C03640=1069.715,413.514,387.232,175.844,35.074,156.512
C03641=1069.725,413.793,387.183,175.850,35.085,156.515
C03642=1069.734,414.072,387.133,175.857,35.096,156.518
C03643=1069.742,414.350,387.084,175.864,35.108,156.520
C03644=1069.751,414.596,387.041,175.870,35.117,156.523
C03645=1069.759,414.842,386.997,175.877,35.127,156.525
C03646=1069.766,415.088,386.953,175.883,35.137,156.527
C03647=1069.774,415.334,386.909,175.888,35.147,156.530
C03648=1069.782,415.580,386.865,175.894,35.157,156.532
C03649=1069.789,415.826,386.822,175.901,35.167,156.535
C03650=1069.797,416.072,386.778,175.907,35.177,156.537
C03651=1069.804,416.319,386.733,175.913,35.187,156.539
C03652=1069.813,416.564,386.689,175.919,35.197,156.542
C03653=1069.820,416.811,386.646,175.926,35.208,156.544
C03654=1069.828,417.056,386.601,175.932,35.218,156.547
C03655=1069.836,417.302,386.557,175.938,35.228,156.549
C03656=1069.844,417.549,386.513,175.944,35.238,156.552
C03657=1069.852,417.794,386.469,175.951,35.248,156.554
C03658=1069.860,418.040,386.425,175.957,35.259,156.557
C03659=1069.868,418.286,386.380,175.963,35.269,156.559
C03660=1069.875,418.532,386.336,175.970,35.279,156.562
C03661=1069.883,418.778,386.292,175.976,35.290,156.564
C03662=1069.892,419.024,386.247,175.983,35.300,156.567
C03663=1069.900,419.270,386.203,175.989,35.310,156.569
C03664=1069.908,419.515,386.159,175.995,35.321,156.572
C03665=1069.916,419.761,386.114,176.003,35.331,156.574
C03666=1069.924,420.007,386.070,176.009,35.342,156.577
C03667=1069.932,420.254,386.025,176.016,35.353,156.579
C03668=1069.940,420.499,385.980,176.022,35.363,156.582
C03669=1069.948,420.745,385.936,176.029,35.373,156.584
C03670=1069.956,420.991,385.892,176.035,35.384,156.587
C03671=1069.964,421.238,385.846,176.042,35.395,156.590
C03672=1069.972,421.483,385.801,176.048,35.406,156.592
C03673=1069.980,421.729,385.757,176.055,35.417,156.595
C03674=1069.988,421.975,385.712,176.062,35.427,156.598
C03675=1069.996,422.220,385.667,176.069,35.438,156.600
C03676=1070.004,422.466,385.622,176.075,35.449,156.603
C03677=1070.012,422.712,385.577,176.082,35.460,156.606
C03678=1070.020,422.957,385.532,176.088,35.471,156.608
C03679=1070.028,423.203,385.487,176.095,35.482,156.611
C03680=1070.037,423.449,385.442,176.102,35.493,156.614
C03681=1070.044,423.695,385.396,176.109,35.504,156.616
C03682=1070.052,423.940,385.352,176.115,35.515,156.619
C03683=1070.061,424.187,385.306,176.122,35.526,156.622
C03684=1070.069,424.432,385.261,176.130,35.537,156.625
C03685=1070.076,424.678,385.216,176.136,35.548,156.627
C03686=1070.085,424.924,385.171,176.143,35.559,156.630
C03687=1070.093,425.169,385.125,176.150,35.571,156.633
C03688=1070.102,425.415,385.080,176.157,35.582,156.636
C03689=1070.110,425.660,385.034,176.164,35.593,156.638
C03690=1070.118,425.907,384.989,176.171,35.604,156.641
C03691=1070.126,426.152,384.944,176.177,35.615,156.644
C03692=1070.135,426.398,384.898,176.185,35.627,156.647
C03693=1070.143,426.643,384.852,176.192,35.638,156.650
C03694=1070.152,426.889,384.807,176.199,35.650,156.652
C03695=1070.159,427.135,384.761,176.206,35.661,156.655
C03696=1070.170,427.431,384.706,176.214,35.675,156.659
C03697=1070.179,427.729,384.650,176.223,35.689,156.662
C03698=1070.190,428.026,384.595,176.232,35.703,156.666
C03699=1070.199,428.324,384.539,176.240,35.717,156.669
C03700=1070.208,428.570,384.493,176.248,35.729,156.672
C03701=1070.217,428.815,384.447,176.255,35.741,156.675
C03702=1070.224,429.061,384.401,176.263,35.753,156.678
C03703=1070.233,429.306,384.355,176.270,35.764,156.681
C03704=1070.241,429.552,384.309,176.277,35.776,156.684
C03705=1070.250,429.797,384.263,176.285,35.788,156.687
C03706=1070.258,430.043,384.217,176.291,35.800,156.690
C03707=1070.267,430.288,384.170,176.299,35.812,156.693
C03708=1070.275,430.534,384.123,176.306,35.824,156.696
C03709=1070.283,430.779,384.078,176.314,35.836,156.699
C03710=1070.292,431.025,384.032,176.321,35.848,156.702
C03711=1070.301,431.270,383.985,176.329,35.860,156.705
C03712=1070.309,431.516,383.939,176.336,35.872,156.708
C03713=1070.318,431.762,383.892,176.344,35.884,156.711
C03714=1070.326,432.007,383.845,176.352,35.896,156.714
C03715=1070.334,432.252,383.799,176.359,35.909,156.717
C03716=1070.343,432.498,383.752,176.367,35.922,156.721
C03717=1070.351,432.743,383.706,176.374,35.934,156.724
C03718=1070.360,432.989,383.659,176.382,35.946,156.727
C03719=1070.368,433.234,383.612,176.390,35.959,156.730
C03720=1070.377,433.479,383.565,176.397,35.971,156.733
C03721=1070.386,433.725,383.518,176.406,35.984,156.736
C03722=1070.393,433.970,383.471,176.414,35.996,156.739
C03723=1070.402,434.216,383.424,176.421,36.009,156.743
C03724=1070.411,434.461,383.377,176.429,36.021,156.746
C03725=1070.419,434.706,383.330,176.437,36.034,156.749
C03726=1070.428,434.952,383.283,176.444,36.047,156.752
C03727=1070.437,435.197,383.236,176.452,36.059,156.756
C03728=1070.445,435.442,383.189,176.461,36.072,156.759
C03729=1070.454,435.687,383.141,176.468,36.085,156.762
C03730=1070.463,435.933,383.095,176.476,36.098,156.765
C03731=1070.471,436.178,383.047,176.484,36.111,156.769
C03732=1070.480,436.423,382.999,176.493,36.124,156.772
C03733=1070.489,436.669,382.952,176.501,36.137,156.775
C03734=1070.498,436.914,382.905,176.508,36.150,156.779
C03735=1070.506,437.159,382.857,176.516,36.163,156.782
C03736=1070.515,437.404,382.810,176.525,36.176,156.785
C03737=1070.525,437.649,382.762,176.533,36.189,156.789
C03738=1070.533,437.894,382.714,176.541,36.202,156.792
C03739=1070.541,438.140,382.667,176.550,36.215,156.796
C03740=1070.551,438.386,382.619,176.558,36.229,156.799
C03741=1070.560,438.630,382.572,176.566,36.242,156.802
C03742=1070.568,438.875,382.523,176.574,36.255,156.806
C03743=1070.578,439.121,382.475,176.582,36.269,156.809
C03744=1070.586,439.365,382.428,176.591,36.282,156.813
C03745=1070.595,439.611,382.380,176.599,36.295,156.816
C03746=1070.604,439.856,382.332,176.608,36.309,156.820
C03747=1070.612,440.101,382.283,176.616,36.323,156.823
C03748=1070.622,440.346,382.236,176.625,36.336,156.827
C03749=1070.631,440.591,382.188,176.633,36.350,156.830
C03750=1070.640,440.837,382.139,176.642,36.364,156.834
C03751=1070.649,441.082,382.092,176.650,36.377,156.838
C03752=1070.657,441.314,382.045,176.659,36.391,156.841
C03753=1070.665,441.548,381.999,176.667,36.404,156.845
C03754=1070.674,441.781,381.953,176.675,36.417,156.848
C03755=1070.683,442.015,381.907,176.683,36.430,156.851
C03756=1070.692,442.248,381.860,176.693,36.444,156.855
C03757=1070.700,442.481,381.814,176.701,36.457,156.858
C03758=1070.708,442.715,381.768,176.709,36.471,156.862
C03759=1070.717,442.948,381.721,176.718,36.484,156.865
C03760=1070.727,443.193,381.673,176.726,36.498,156.869
C03761=1070.736,443.438,381.624,176.735,36.513,156.873
C03762=1070.745,443.682,381.575,176.744,36.527,156.877
C03763=1070.754,443.927,381.526,176.754,36.541,156.881
C03764=1070.764,444.172,381.478,176.762,36.556,156.884
C03765=1070.773,444.418,381.429,176.771,36.570,156.888
C03766=1070.781,444.662,381.380,176.781,36.584,156.892
C03767=1070.790,444.908,381.331,176.790,36.599,156.896
C03768=1070.800,445.152,381.281,176.799,36.614,156.900
C03769=1070.809,445.397,381.232,176.808,36.628,156.904
C03770=1070.819,445.642,381.183,176.817,36.643,156.907
C03771=1070.828,445.887,381.133,176.826,36.658,156.911
C03772=1070.837,446.132,381.085,176.836,36.672,156.915
C03773=1070.846,446.376,381.035,176.845,36.687,156.919
C03774=1070.855,446.621,380.986,176.855,36.702,156.923
C03775=1070.864,446.866,380.936,176.864,36.717,156.927
C03776=1070.874,447.111,380.887,176.874,36.732,156.931
C03777=1070.884,447.355,380.837,176.883,36.747,156.935
C03778=1070.893,447.601,380.788,176.893,36.762,156.939
C03779=1070.903,447.846,380.738,176.902,36.777,156.943
C03780=1070.913,448.089,380.688,176.911,36.793,156.947
C03781=1070.922,448.332,380.640,176.920,36.807,156.951
C03782=1070.932,448.577,380.590,176.929,36.822,156.955
C03783=1070.944,448.821,380.542,176.937,36.836,156.959
C03784=1070.957,449.066,380.495,176.945,36.850,156.963
C03785=1070.972,449.311,380.449,176.953,36.863,156.966
C03786=1070.987,449.556,380.402,176.960,36.876,156.970
C03787=1071.004,449.802,380.357,176.968,36.888,156.973
C03788=1070.654,449.802,380.106,176.954,37.029,157.010
C03789=1070.638,449.556,380.151,176.947,37.016,157.007
C03790=1070.622,449.311,380.197,176.939,37.004,157.004
C03791=1070.608,449.066,380.244,176.931,36.990,157.000
C03792=1070.595,448.821,380.291,176.923,36.977,156.996
C03793=1070.582,448.576,380.339,176.914,36.963,156.993
C03794=1070.571,448.332,380.388,176.905,36.948,156.989
C03795=1070.562,448.088,380.437,176.896,36.933,156.985
C03796=1070.553,447.845,380.487,176.886,36.918,156.981
C03797=1070.543,447.601,380.537,176.877,36.903,156.977
C03798=1070.533,447.356,380.587,176.867,36.888,156.973
C03799=1070.523,447.111,380.636,176.858,36.873,156.969
C03800=1070.514,446.866,380.685,176.848,36.858,156.965
C03801=1070.505,446.621,380.735,176.838,36.843,156.961
C03802=1070.496,446.376,380.785,176.829,36.828,156.957
C03803=1070.486,446.131,380.834,176.819,36.814,156.953
C03804=1070.477,445.887,380.884,176.810,36.799,156.949
C03805=1070.468,445.641,380.933,176.800,36.784,156.945
C03806=1070.458,445.397,380.982,176.792,36.770,156.941
C03807=1070.449,445.153,381.031,176.782,36.755,156.937
C03808=1070.440,444.908,381.080,176.773,36.741,156.933
C03809=1070.431,444.663,381.130,176.764,36.726,156.929
C03810=1070.422,444.417,381.179,176.754,36.711,156.925
C03811=1070.412,444.173,381.228,176.745,36.697,156.922
C03812=1070.403,443.928,381.277,176.736,36.683,156.918
C03813=1070.394,443.683,381.326,176.727,36.668,156.914
C03814=1070.384,443.438,381.374,176.718,36.654,156.910
C03815=1070.375,443.193,381.423,176.708,36.640,156.906
C03816=1070.366,442.949,381.472,176.700,36.626,156.903
C03817=1070.358,442.724,381.516,176.692,36.612,156.899
C03818=1070.349,442.500,381.561,176.684,36.600,156.896
C03819=1070.341,442.276,381.606,176.675,36.587,156.892
C03820=1070.333,442.052,381.649,176.667,36.574,156.889
C03821=1070.324,441.828,381.694,176.659,36.562,156.886
C03822=1070.316,441.604,381.739,176.651,36.549,156.882
C03823=1070.308,441.380,381.782,176.643,36.536,156.879
C03824=1070.300,441.156,381.827,176.635,36.524,156.876
C03825=1070.291,440.912,381.876,176.627,36.510,156.872
C03826=1070.282,440.666,381.924,176.618,36.496,156.869
C03827=1070.273,440.421,381.973,176.609,36.482,156.865
C03828=1070.264,440.176,382.020,176.600,36.468,156.861
C03829=1070.254,439.931,382.069,176.592,36.455,156.858
C03830=1070.246,439.686,382.117,176.583,36.442,156.854
C03831=1070.237,439.441,382.164,176.575,36.428,156.851
C03832=1070.228,439.195,382.213,176.566,36.415,156.847
C03833=1070.219,438.951,382.261,176.558,36.401,156.844
C03834=1070.210,438.705,382.308,176.549,36.388,156.840
C03835=1070.202,438.460,382.357,176.541,36.374,156.837
C03836=1070.193,438.215,382.404,176.533,36.361,156.833
C03837=1070.183,437.969,382.452,176.524,36.348,156.830
C03838=1070.174,437.724,382.499,176.516,36.335,156.827
C03839=1070.166,437.480,382.547,176.507,36.322,156.823
C03840=1070.157,437.234,382.595,176.499,36.309,156.820
C03841=1070.148,436.989,382.643,176.491,36.296,156.817
C03842=1070.139,436.744,382.690,176.483,36.283,156.813
C03843=1070.130,436.498,382.737,176.475,36.270,156.810
C03844=1070.121,436.253,382.785,176.467,36.257,156.807
C03845=1070.112,436.008,382.832,176.459,36.244,156.803
C03846=1070.104,435.762,382.879,176.450,36.231,156.800
C03847=1070.096,435.517,382.927,176.442,36.218,156.797
C03848=1070.087,435.272,382.974,176.434,36.205,156.793
C03849=1070.078,435.027,383.021,176.427,36.193,156.790
C03850=1070.069,434.781,383.069,176.419,36.180,156.787
C03851=1070.060,434.536,383.115,176.410,36.167,156.784
C03852=1070.051,434.291,383.163,176.402,36.155,156.780
C03853=1070.043,434.045,383.210,176.395,36.142,156.777
C03854=1070.034,433.800,383.256,176.387,36.130,156.774
C03855=1070.026,433.554,383.303,176.379,36.117,156.771
C03856=1070.017,433.309,383.351,176.371,36.105,156.768
C03857=1070.008,433.064,383.397,176.364,36.092,156.764
C03858=1070.001,432.818,383.445,176.356,36.080,156.761
C03859=1069.992,432.572,383.491,176.348,36.068,156.758
C03860=1069.984,432.328,383.538,176.341,36.055,156.755
C03861=1069.976,432.082,383.584,176.333,36.043,156.752
C03862=1069.967,431.837,383.631,176.325,36.031,156.749
C03863=1069.958,431.591,383.678,176.318,36.018,156.746
C03864=1069.950,431.346,383.725,176.310,36.006,156.743
C03865=1069.941,431.100,383.771,176.303,35.994,156.740
C03866=1069.932,430.855,383.817,176.295,35.982,156.737
C03867=1069.924,430.609,383.863,176.287,35.970,156.734
C03868=1069.916,430.364,383.910,176.280,35.958,156.730
C03869=1069.907,430.118,383.957,176.272,35.946,156.727
C03870=1069.898,429.873,384.002,176.265,35.934,156.724
C03871=1069.890,429.627,384.049,176.257,35.923,156.721
C03872=1069.882,429.382,384.095,176.250,35.910,156.718
C03873=1069.874,429.136,384.141,176.242,35.899,156.716
C03874=1069.865,428.891,384.188,176.235,35.887,156.713
C03875=1069.857,428.645,384.233,176.228,35.875,156.710
C03876=1069.849,428.399,384.279,176.221,35.864,156.707
C03877=1069.838,428.100,384.335,176.212,35.849,156.703
C03878=1069.829,427.801,384.391,176.203,35.835,156.700
C03879=1069.818,427.503,384.447,176.194,35.821,156.696
C03880=1069.808,427.203,384.503,176.185,35.807,156.693
C03881=1069.800,426.957,384.549,176.178,35.796,156.690
C03882=1069.791,426.712,384.594,176.171,35.784,156.687
C03883=1069.783,426.466,384.640,176.164,35.773,156.684
C03884=1069.775,426.220,384.685,176.156,35.761,156.681
C03885=1069.766,425.974,384.731,176.150,35.750,156.678
C03886=1069.758,425.729,384.776,176.142,35.739,156.676
C03887=1069.750,425.483,384.822,176.135,35.728,156.673
C03888=1069.741,425.238,384.867,176.129,35.716,156.670
C03889=1069.733,424.992,384.913,176.121,35.705,156.667
C03890=1069.725,424.747,384.958,176.114,35.694,156.665
C03891=1069.717,424.501,385.004,176.108,35.683,156.662
C03892=1069.709,424.255,385.049,176.101,35.672,156.659
C03893=1069.701,424.009,385.094,176.093,35.661,156.656
C03894=1069.692,423.764,385.140,176.087,35.650,156.654
C03895=1069.685,423.517,385.185,176.080,35.639,156.651
C03896=1069.676,423.272,385.230,176.073,35.628,156.648
C03897=1069.667,423.027,385.275,176.066,35.617,156.645
C03898=1069.660,422.780,385.320,176.060,35.606,156.643
C03899=1069.652,422.535,385.365,176.053,35.595,156.640
C03900=1069.644,422.289,385.410,176.045,35.584,156.637
C03901=1069.635,422.043,385.455,176.039,35.573,156.635
C03902=1069.628,421.797,385.500,176.032,35.563,156.632
C03903=1069.620,421.552,385.545,176.026,35.552,156.629
C03904=1069.611,421.306,385.590,176.019,35.541,156.627
C03905=1069.604,421.060,385.635,176.012,35.530,156.624
C03906=1069.595,420.814,385.679,176.005,35.520,156.622
C03907=1069.587,420.568,385.724,175.999,35.509,156.619
C03908=1069.579,420.322,385.768,175.993,35.499,156.616
C03909=1069.571,420.076,385.813,175.986,35.488,156.614
C03910=1069.563,419.831,385.858,175.980,35.477,156.611
C03911=1069.555,419.585,385.903,175.973,35.467,156.609
C03912=1069.547,419.339,385.947,175.966,35.457,156.606
C03913=1069.539,419.093,385.991,175.959,35.446,156.604
C03914=1069.530,418.846,386.035,175.953,35.436,156.601
C03915=1069.522,418.601,386.080,175.947,35.426,156.599
C03916=1069.515,418.355,386.125,175.940,35.416,156.596
C03917=1069.507,418.109,386.169,175.934,35.405,156.594
C03918=1069.499,417.863,386.213,175.928,35.395,156.591
C03919=1069.491,417.617,386.258,175.921,35.384,156.589
C03920=1069.483,417.371,386.301,175.915,35.374,156.586
C03921=1069.475,417.125,386.346,175.909,35.364,156.584
C03922=1069.467,416.879,386.390,175.902,35.354,156.581
C03923=1069.459,416.633,386.434,175.896,35.344,156.579
C03924=1069.451,416.387,386.478,175.890,35.334,156.576
C03925=1069.444,416.141,386.523,175.883,35.323,156.574
C03926=1069.437,415.896,386.566,175.876,35.313,156.571
C03927=1069.429,415.650,386.610,175.870,35.304,156.569
C03928=1069.421,415.404,386.654,175.864,35.293,156.567
C03929=1069.413,415.158,386.698,175.859,35.284,156.564
C03930=1069.405,414.911,386.742,175.851,35.274,156.562
C03931=1069.397,414.665,386.786,175.846,35.264,156.560
C03932=1069.389,414.419,386.830,175.840,35.254,156.557
C03933=1069.380,414.139,386.879,175.832,35.243,156.554
C03934=1069.371,413.859,386.929,175.825,35.232,156.552
C03935=1069.362,413.579,386.979,175.818,35.220,156.549
C03936=1069.353,413.298,387.028,175.811,35.210,156.546
C03937=1069.346,413.053,387.072,175.805,35.200,156.544
C03938=1069.337,412.807,387.115,175.799,35.190,156.542
C03939=1069.329,412.561,387.158,175.793,35.180,156.540
C03940=1069.322,412.314,387.202,175.788,35.171,156.537
C03941=1069.314,412.069,387.245,175.782,35.162,156.535
C03942=1069.306,411.823,387.288,175.776,35.152,156.533
C03943=1069.298,411.576,387.332,175.770,35.142,156.530
C03944=1069.290,411.330,387.375,175.764,35.133,156.528
C03945=1069.284,411.084,387.418,175.757,35.123,156.526
C03946=1069.275,410.838,387.461,175.751,35.113,156.524
C03947=1069.267,410.591,387.505,175.745,35.104,156.521
C03948=1069.260,410.346,387.548,175.740,35.095,156.519
C03949=1069.252,410.099,387.591,175.734,35.085,156.517
C03950=1069.245,409.853,387.633,175.728,35.076,156.515
C03951=1069.237,409.607,387.677,175.722,35.067,156.513
C03952=1069.230,409.361,387.720,175.716,35.057,156.510
C03953=1069.222,409.115,387.763,175.710,35.048,156.508
C03954=1069.214,408.868,387.806,175.704,35.039,156.506
C03955=1069.207,408.622,387.849,175.699,35.030,156.504
C03956=1069.199,408.376,387.892,175.693,35.020,156.502
C03957=1069.191,408.130,387.935,175.687,35.011,156.499
C03958=1069.184,407.884,387.977,175.682,35.002,156.497
C03959=1069.176,407.637,388.020,175.676,34.993,156.495
C03960=1069.169,407.392,388.063,175.671,34.984,156.493
C03961=1069.161,407.145,388.105,175.665,34.975,156.491
C03962=1069.154,406.899,388.149,175.659,34.966,156.489
C03963=1069.146,406.652,388.192,175.653,34.956,156.486
C03964=1069.139,406.406,388.234,175.648,34.948,156.484
C03965=1069.132,406.161,388.277,175.642,34.938,156.482
C03966=1069.123,405.914,388.319,175.636,34.930,156.480
C03967=1069.117,405.668,388.362,175.631,34.921,156.478
C03968=1069.109,405.422,388.404,175.626,34.912,156.476
C03969=1069.102,405.175,388.446,175.620,34.903,156.474
C03970=1069.094,404.929,388.488,175.614,34.894,156.472
C03971=1069.086,404.683,388.530,175.608,34.885,156.470
C03972=1069.079,404.436,388.573,175.603,34.876,156.468
C03973=1069.071,404.190,388.615,175.598,34.868,156.466
C03974=1069.064,403.943,388.658,175.592,34.859,156.464
C03975=1069.056,403.697,388.700,175.587,34.850,156.462
C03976=1069.049,403.451,388.742,175.581,34.841,156.460
C03977=1069.042,403.204,388.785,175.575,34.833,156.458
C03978=1069.034,402.959,388.827,175.570,34.824,156.455
C03979=1069.027,402.713,388.868,175.565,34.815,156.453
C03980=1069.018,402.466,388.911,175.559,34.807,156.451
C03981=1069.012,402.219,388.953,175.553,34.798,156.449
C03982=1069.004,401.973,388.995,175.549,34.790,156.447
C03983=1068.997,401.727,389.036,175.543,34.781,156.445
C03984=1068.989,401.481,389.078,175.537,34.773,156.444
C03985=1068.981,401.234,389.120,175.532,34.764,156.442
C03986=1068.974,400.987,389.163,175.527,34.756,156.440
C03987=1068.967,400.741,389.204,175.521,34.747,156.438
C03988=1068.959,400.495,389.246,175.516,34.739,156.436
C03989=1068.951,400.219,389.293,175.510,34.729,156.434
C03990=1068.943,399.942,389.339,175.504,34.719,156.431
C03991=1068.935,399.666,389.386,175.498,34.710,156.429
C03992=1068.926,399.390,389.433,175.492,34.701,156.427
C03993=1068.919,399.143,389.474,175.487,34.693,156.425
C03994=1068.912,398.897,389.516,175.482,34.684,156.423
C03995=1068.904,398.651,389.558,175.476,34.676,156.421
C03996=1068.897,398.404,389.599,175.472,34.668,156.419
C03997=1068.889,398.158,389.641,175.466,34.660,156.417
C03998=1068.882,397.912,389.682,175.460,34.651,156.416
C03999=1068.875,397.665,389.723,175.456,34.643,156.414
C04000=1068.867,397.418,389.765,175.450,34.635,156.412
C04001=1068.860,397.172,389.806,175.445,34.627,156.410
C04002=1068.853,396.926,389.848,175.440,34.618,156.408
C04003=1068.846,396.680,389.889,175.434,34.611,156.406
C04004=1068.839,396.433,389.930,175.430,34.602,156.404
C04005=1068.831,396.187,389.971,175.424,34.594,156.402
C04006=1068.824,395.940,390.012,175.420,34.586,156.401
C04007=1068.817,395.694,390.053,175.414,34.578,156.399
C04008=1068.809,395.447,390.095,175.409,34.570,156.397
C04009=1068.801,395.201,390.135,175.404,34.562,156.395
C04010=1068.795,394.955,390.176,175.399,34.554,156.393
C04011=1068.787,394.708,390.217,175.394,34.546,156.391
C04012=1068.780,394.462,390.259,175.389,34.538,156.390
C04013=1068.773,394.215,390.300,175.384,34.531,156.388
C04014=1068.766,393.969,390.341,175.378,34.522,156.386
C04015=1068.759,393.722,390.381,175.374,34.515,156.384
C04016=1068.751,393.476,390.422,175.368,34.507,156.383
C04017=1068.744,393.229,390.463,175.364,34.499,156.381
C04018=1068.737,392.983,390.504,175.358,34.491,156.379
C04019=1068.730,392.736,390.545,175.353,34.484,156.377
C04020=1068.722,392.490,390.585,175.348,34.476,156.376
C04021=1068.716,392.244,390.626,175.343,34.468,156.374
C04022=1068.709,391.997,390.667,175.338,34.460,156.372
C04023=1068.701,391.750,390.707,175.334,34.453,156.370
C04024=1068.694,391.504,390.748,175.328,34.445,156.369
C04025=1068.687,391.257,390.789,175.324,34.437,156.367
C04026=1068.679,391.011,390.829,175.318,34.429,156.365
C04027=1068.672,390.764,390.869,175.314,34.422,156.363
C04028=1068.665,390.518,390.911,175.309,34.414,156.362
C04029=1068.658,390.272,390.950,175.304,34.407,156.360
C04030=1068.651,390.025,390.991,175.299,34.399,156.358
C04031=1068.643,389.778,391.031,175.294,34.392,156.356
C04032=1068.637,389.532,391.071,175.289,34.384,156.355
C04033=1068.629,389.285,391.112,175.284,34.376,156.353
C04034=1068.622,389.039,391.152,175.279,34.369,156.351
C04035=1068.615,388.792,391.192,175.274,34.361,156.350
C04036=1068.607,388.546,391.232,175.270,34.354,156.348
C04037=1068.600,388.299,391.273,175.264,34.346,156.346
C04038=1068.592,388.052,391.313,175.260,34.339,156.345
C04039=1068.586,387.806,391.353,175.255,34.332,156.343
C04040=1068.579,387.559,391.392,175.250,34.325,156.341
C04041=1068.571,387.313,391.432,175.246,34.317,156.340
C04042=1068.564,387.067,391.473,175.240,34.310,156.338
C04043=1068.557,386.820,391.513,175.236,34.302,156.337
C04044=1068.550,386.573,391.553,175.231,34.295,156.335
C04045=1068.542,386.313,391.595,175.226,34.287,156.333
C04046=1068.535,386.052,391.637,175.221,34.279,156.331
C04047=1068.528,385.792,391.680,175.216,34.272,156.330
C04048=1068.521,385.532,391.722,175.211,34.264,156.328
C04049=1068.513,385.285,391.761,175.206,34.257,156.326
C04050=1068.506,385.038,391.801,175.201,34.250,156.325
C04051=1068.499,384.792,391.841,175.197,34.243,156.323
C04052=1068.492,384.546,391.881,175.192,34.235,156.322
C04053=1068.485,384.301,391.921,175.188,34.228,156.320
C04054=1068.478,384.056,391.959,175.182,34.221,156.318
C04055=1068.471,383.811,391.999,175.178,34.214,156.317
C04056=1068.464,383.567,392.038,175.174,34.207,156.315
C04057=1068.458,383.322,392.078,175.168,34.200,156.314
C04058=1068.450,383.078,392.117,175.164,34.193,156.312
C04059=1068.444,382.833,392.156,175.160,34.186,156.311
C04060=1068.436,382.588,392.196,175.155,34.179,156.309
C04061=1068.430,382.342,392.236,175.151,34.171,156.307
C04062=1068.423,382.095,392.275,175.146,34.165,156.306
C04063=1068.416,381.849,392.314,175.141,34.157,156.304
C04064=1068.409,381.601,392.354,175.137,34.151,156.303
C04065=1068.402,381.355,392.393,175.132,34.143,156.301
C04066=1068.396,381.108,392.432,175.127,34.137,156.300
C04067=1068.388,380.862,392.472,175.123,34.129,156.298
C04068=1068.381,380.614,392.511,175.118,34.123,156.297
C04069=1068.374,380.368,392.551,175.114,34.116,156.295
C04070=1068.367,380.121,392.589,175.109,34.109,156.294
C04071=1068.360,379.874,392.628,175.104,34.102,156.292
C04072=1068.353,379.628,392.668,175.100,34.095,156.291
C04073=1068.346,379.381,392.707,175.096,34.088,156.289
C04074=1068.339,379.134,392.746,175.090,34.081,156.288
C04075=1068.332,378.888,392.785,175.086,34.075,156.286
C04076=1068.325,378.641,392.824,175.082,34.068,156.285
C04077=1068.318,378.394,392.863,175.077,34.061,156.283
C04078=1068.311,378.147,392.902,175.073,34.054,156.282
C04079=1068.305,377.900,392.941,175.068,34.048,156.280
C04080=1068.297,377.654,392.980,175.064,34.041,156.279
C04081=1068.290,377.407,393.020,175.059,34.034,156.277
C04082=1068.283,377.160,393.058,175.055,34.027,156.276
C04083=1068.276,376.913,393.097,175.051,34.021,156.274
C04084=1068.270,376.666,393.136,175.046,34.014,156.273
C04085=1068.263,376.419,393.175,175.041,34.007,156.271
C04086=1068.256,376.172,393.214,175.037,34.001,156.270
C04087=1068.249,375.926,393.253,175.032,33.994,156.268
C04088=1068.242,375.679,393.291,175.028,33.987,156.267
C04089=1068.236,375.432,393.330,175.024,33.981,156.266
C04090=1068.229,375.185,393.369,175.020,33.974,156.264
C04091=1068.222,374.938,393.408,175.015,33.967,156.263
C04092=1068.215,374.691,393.446,175.011,33.961,156.261
C04093=1068.209,374.444,393.485,175.007,33.954,156.260
C04094=1068.202,374.197,393.524,175.001,33.947,156.258
C04095=1068.195,373.951,393.562,174.997,33.941,156.257
C04096=1068.188,373.705,393.600,174.993,33.934,156.256
C04097=1068.182,373.464,393.638,174.989,33.928,156.254
C04098=1068.175,373.223,393.676,174.984,33.922,156.253
C04099=1068.169,372.983,393.714,174.980,33.915,156.251
C04100=1068.162,372.742,393.750,174.976,33.909,156.250
C04101=1068.155,372.501,393.788,174.972,33.903,156.249
C04102=1068.148,372.261,393.825,174.967,33.896,156.247
C04103=1068.141,372.020,393.862,174.963,33.890,156.246
C04104=1068.135,371.780,393.900,174.959,33.884,156.245
C04105=1068.128,371.533,393.938,174.955,33.878,156.243
C04106=1068.121,371.286,393.976,174.950,33.871,156.242
C04107=1068.114,371.039,394.014,174.946,33.865,156.241
C04108=1068.107,370.792,394.053,174.942,33.859,156.239
C04109=1068.101,370.545,394.091,174.938,33.853,156.238
C04110=1068.093,370.298,394.129,174.933,33.846,156.237
C04111=1068.087,370.051,394.167,174.929,33.840,156.235
C04112=1068.080,369.805,394.205,174.925,33.833,156.234
C04113=1068.073,369.558,394.243,174.921,33.827,156.232
C04114=1068.067,369.310,394.281,174.917,33.821,156.231
C04115=1068.059,369.064,394.320,174.912,33.814,156.230
C04116=1068.053,368.816,394.358,174.908,33.808,156.228
C04117=1068.046,368.570,394.395,174.904,33.802,156.227
C04118=1068.040,368.322,394.433,174.900,33.796,156.226
C04119=1068.033,368.076,394.472,174.895,33.790,156.224
C04120=1068.026,367.828,394.509,174.891,33.784,156.223
C04121=1068.020,367.582,394.547,174.887,33.777,156.222
C04122=1068.012,367.335,394.585,174.883,33.771,156.220
C04123=1068.006,367.087,394.623,174.879,33.765,156.219
C04124=1067.999,366.841,394.660,174.874,33.758,156.218
C04125=1067.992,366.594,394.699,174.870,33.753,156.217
C04126=1067.985,366.347,394.736,174.866,33.746,156.215
C04127=1067.979,366.100,394.774,174.862,33.740,156.214
C04128=1067.972,365.853,394.812,174.857,33.734,156.213
C04129=1067.966,365.605,394.850,174.853,33.728,156.211
C04130=1067.959,365.359,394.887,174.849,33.722,156.210
C04131=1067.952,365.112,394.925,174.845,33.715,156.209
C04132=1067.946,364.865,394.962,174.841,33.710,156.207
C04133=1067.939,364.618,395.000,174.838,33.703,156.206
C04134=1067.932,364.370,395.037,174.833,33.698,156.205
C04135=1067.926,364.123,395.075,174.829,33.691,156.204
C04136=1067.919,363.876,395.112,174.825,33.686,156.202
C04137=1067.912,363.629,395.150,174.821,33.679,156.201
C04138=1067.906,363.382,395.188,174.817,33.674,156.200
C04139=1067.899,363.135,395.225,174.812,33.667,156.198
C04140=1067.892,362.888,395.262,174.808,33.662,156.197
C04141=1067.885,362.641,395.299,174.804,33.656,156.196
C04142=1067.879,362.394,395.337,174.800,33.649,156.195
C04143=1067.872,362.146,395.374,174.796,33.644,156.193
C04144=1067.865,361.899,395.411,174.793,33.638,156.192
C04145=1067.858,361.653,395.448,174.788,33.632,156.191
C04146=1067.852,361.405,395.486,174.784,33.626,156.190
C04147=1067.846,361.158,395.523,174.780,33.620,156.188
C04148=1067.839,360.910,395.560,174.776,33.614,156.187
C04149=1067.832,360.664,395.597,174.772,33.609,156.186
C04150=1067.825,360.417,395.634,174.768,33.603,156.185
C04151=1067.819,360.170,395.671,174.763,33.596,156.184
C04152=1067.812,359.922,395.709,174.760,33.591,156.182
C04153=1067.805,359.692,395.743,174.756,33.586,156.181
C04154=1067.800,359.463,395.777,174.752,33.580,156.180
C04155=1067.794,359.233,395.811,174.749,33.575,156.179
C04156=1067.788,359.003,395.846,174.745,33.569,156.178
C04157=1067.782,358.773,395.881,174.742,33.564,156.177
C04158=1067.776,358.543,395.915,174.737,33.558,156.176
C04159=1067.769,358.313,395.949,174.733,33.553,156.174
C04160=1067.763,358.084,395.984,174.730,33.548,156.173
C04161=1067.757,357.837,396.021,174.726,33.542,156.172
C04162=1067.750,357.589,396.057,174.722,33.536,156.171
C04163=1067.743,357.342,396.094,174.718,33.531,156.170
C04164=1067.736,357.095,396.131,174.715,33.525,156.169
C04165=1067.730,356.848,396.168,174.710,33.519,156.167
C04166=1067.723,356.600,396.204,174.706,33.514,156.166
C04167=1067.717,356.353,396.241,174.702,33.508,156.165
C04168=1067.710,356.106,396.277,174.698,33.502,156.164
C04169=1067.703,355.858,396.314,174.695,33.497,156.163
C04170=1067.697,355.611,396.351,174.691,33.491,156.162
C04171=1067.690,355.364,396.388,174.687,33.485,156.160
C04172=1067.684,355.117,396.424,174.683,33.480,156.159
C04173=1067.677,354.870,396.461,174.678,33.474,156.158
C04174=1067.671,354.623,396.498,174.675,33.469,156.157
C04175=1067.664,354.375,396.534,174.671,33.463,156.156
C04176=1067.657,354.128,396.570,174.667,33.457,156.154
C04177=1067.650,353.881,396.607,174.663,33.452,156.153
C04178=1067.644,353.634,396.643,174.660,33.446,156.152
C04179=1067.638,353.387,396.680,174.656,33.440,156.151
C04180=1067.631,353.139,396.716,174.652,33.435,156.150
C04181=1067.624,352.892,396.753,174.647,33.429,156.149
C04182=1067.618,352.644,396.789,174.644,33.424,156.148
C04183=1067.612,352.397,396.825,174.640,33.418,156.146
C04184=1067.605,352.150,396.862,174.636,33.413,156.145
C04185=1067.599,351.903,396.898,174.633,33.407,156.144
C04186=1067.592,351.656,396.934,174.629,33.402,156.143
C04187=1067.586,351.408,396.970,174.625,33.397,156.142
C04188=1067.579,351.161,397.006,174.621,33.391,156.141
C04189=1067.572,350.913,397.043,174.618,33.386,156.140
C04190=1067.565,350.667,397.079,174.613,33.380,156.138
C04191=1067.559,350.419,397.115,174.609,33.374,156.137
C04192=1067.553,350.172,397.151,174.605,33.369,156.136
C04193=1067.546,349.924,397.186,174.602,33.364,156.135
C04194=1067.539,349.677,397.223,174.598,33.358,156.134
C04195=1067.533,349.430,397.260,174.594,33.353,156.133
C04196=1067.526,349.182,397.295,174.591,33.348,156.132
C04197=1067.520,348.935,397.331,174.587,33.342,156.131
C04198=1067.514,348.688,397.367,174.583,33.337,156.130
C04199=1067.507,348.440,397.403,174.580,33.331,156.129
C04200=1067.501,348.193,397.438,174.576,33.326,156.127
C04201=1067.494,347.946,397.475,174.571,33.321,156.126
C04202=1067.488,347.698,397.511,174.568,33.316,156.125
C04203=1067.481,347.451,397.547,174.564,33.310,156.124
C04204=1067.475,347.203,397.583,174.560,33.304,156.123
C04205=1067.467,346.957,397.618,174.557,33.299,156.122
C04206=1067.461,346.709,397.654,174.553,33.294,156.121
C04207=1067.455,346.461,397.690,174.549,33.289,156.120
C04208=1067.448,346.214,397.726,174.546,33.283,156.119
C04209=1067.442,345.986,397.758,174.542,33.279,156.118
C04210=1067.436,345.758,397.791,174.539,33.273,156.117
C04211=1067.431,345.531,397.824,174.536,33.269,156.116
C04212=1067.425,345.303,397.857,174.532,33.264,156.115
C04213=1067.419,345.074,397.890,174.529,33.259,156.114
C04214=1067.413,344.846,397.922,174.525,33.254,156.113
C04215=1067.407,344.619,397.956,174.521,33.249,156.112
C04216=1067.401,344.390,397.988,174.518,33.245,156.111
C04217=1067.395,344.143,398.024,174.514,33.239,156.110
C04218=1067.388,343.895,398.059,174.511,33.234,156.109
C04219=1067.382,343.648,398.095,174.507,33.229,156.108
C04220=1067.375,343.400,398.130,174.504,33.224,156.107
C04221=1067.368,343.154,398.166,174.500,33.218,156.105
C04222=1067.363,342.907,398.201,174.496,33.213,156.104
C04223=1067.356,342.659,398.236,174.493,33.208,156.103
C04224=1067.349,342.412,398.272,174.489,33.203,156.102
C04225=1067.343,342.164,398.307,174.486,33.198,156.101
C04226=1067.336,341.917,398.342,174.482,33.192,156.100
C04227=1067.330,341.670,398.378,174.478,33.188,156.099
C04228=1067.324,341.422,398.413,174.475,33.182,156.098
C04229=1067.317,341.175,398.448,174.471,33.177,156.097
C04230=1067.310,340.927,398.483,174.468,33.172,156.096
C04231=1067.304,340.679,398.519,174.464,33.167,156.095
C04232=1067.298,340.431,398.554,174.460,33.162,156.094
C04233=1067.291,340.184,398.589,174.456,33.157,156.093
C04234=1067.285,339.937,398.624,174.452,33.152,156.092
C04235=1067.279,339.690,398.659,174.449,33.146,156.091
C04236=1067.272,339.442,398.694,174.445,33.142,156.090
C04237=1067.265,339.194,398.729,174.442,33.136,156.089
C04238=1067.259,338.947,398.765,174.438,33.132,156.088
C04239=1067.253,338.699,398.800,174.435,33.126,156.087
C04240=1067.246,338.453,398.834,174.431,33.121,156.086
C04241=1067.241,338.204,398.870,174.428,33.116,156.085
C04242=1067.234,337.957,398.905,174.424,33.111,156.084
C04243=1067.227,337.710,398.940,174.421,33.106,156.083
C04244=1067.221,337.462,398.974,174.417,33.101,156.082
C04245=1067.215,337.215,399.009,174.414,33.096,156.081
C04246=1067.208,336.967,399.045,174.410,33.091,156.080
C04247=1067.202,336.719,399.079,174.407,33.086,156.079
C04248=1067.195,336.472,399.114,174.403,33.081,156.078
C04249=1067.189,336.225,399.148,174.400,33.076,156.077
C04250=1067.183,335.977,399.183,174.396,33.071,156.076
C04251=1067.176,335.729,399.218,174.393,33.066,156.075
C04252=1067.169,335.482,399.253,174.389,33.061,156.074
C04253=1067.164,335.235,399.287,174.386,33.057,156.073
C04254=1067.157,334.987,399.322,174.382,33.051,156.072
C04255=1067.150,334.739,399.357,174.379,33.047,156.071
C04256=1067.144,334.492,399.392,174.375,33.042,156.070
C04257=1067.138,334.245,399.426,174.372,33.037,156.069
C04258=1067.131,333.997,399.460,174.368,33.032,156.068
C04259=1067.124,333.749,399.495,174.365,33.027,156.067
C04260=1067.119,333.502,399.529,174.361,33.022,156.066
C04261=1067.112,333.254,399.564,174.357,33.017,156.065
C04262=1067.105,333.007,399.599,174.353,33.012,156.064
C04263=1067.099,332.759,399.633,174.350,33.007,156.063
C04264=1067.093,332.511,399.667,174.347,33.003,156.062
C04265=1067.088,332.281,399.700,174.343,32.998,156.061
C04266=1067.081,332.051,399.732,174.340,32.993,156.060
C04267=1067.076,331.820,399.764,174.337,32.989,156.060
C04268=1067.070,331.590,399.796,174.334,32.984,156.059
C04269=1067.064,331.360,399.828,174.331,32.980,156.058
C04270=1067.058,331.129,399.860,174.327,32.975,156.057
C04271=1067.052,330.899,399.891,174.324,32.971,156.056
C04272=1067.046,330.668,399.924,174.321,32.966,156.055
C04273=1067.040,330.421,399.957,174.318,32.962,156.054
C04274=1067.033,330.173,399.992,174.314,32.957,156.053
C04275=1067.027,329.925,400.026,174.311,32.952,156.052
C04276=1067.020,329.679,400.060,174.307,32.947,156.051
C04277=1067.013,329.431,400.095,174.304,32.943,156.050
C04278=1067.007,329.183,400.129,174.300,32.938,156.049
C04279=1067.000,328.936,400.162,174.297,32.933,156.048
C04280=1066.994,328.687,400.196,174.294,32.928,156.048
C04281=1066.988,328.440,400.230,174.290,32.924,156.047
C04282=1066.981,328.192,400.264,174.287,32.919,156.046
C04283=1066.975,327.944,400.298,174.283,32.915,156.045
C04284=1066.968,327.697,400.332,174.280,32.910,156.044
C04285=1066.962,327.449,400.366,174.277,32.905,156.043
C04286=1066.956,327.202,400.400,174.273,32.900,156.042
C04287=1066.949,326.954,400.434,174.270,32.895,156.041
C04288=1066.943,326.707,400.468,174.266,32.891,156.040
C04289=1066.936,326.459,400.501,174.263,32.886,156.039
C04290=1066.930,326.212,400.535,174.260,32.882,156.038
C04291=1066.923,325.964,400.569,174.256,32.877,156.037
C04292=1066.917,325.717,400.603,174.253,32.872,156.037
C04293=1066.910,325.469,400.638,174.250,32.867,156.036
C04294=1066.904,325.221,400.671,174.246,32.863,156.035
C04295=1066.898,324.973,400.705,174.243,32.858,156.034
C04296=1066.891,324.726,400.738,174.240,32.854,156.033
C04297=1066.886,324.478,400.772,174.236,32.849,156.032
C04298=1066.878,324.230,400.806,174.233,32.844,156.031
C04299=1066.872,323.983,400.840,174.230,32.840,156.030
C04300=1066.866,323.735,400.873,174.226,32.835,156.029
C04301=1066.860,323.488,400.907,174.223,32.830,156.028
C04302=1066.854,323.240,400.941,174.221,32.826,156.027
C04303=1066.847,322.992,400.974,174.217,32.821,156.027
C04304=1066.841,322.745,401.008,174.214,32.817,156.026
C04305=1066.834,322.496,401.041,174.211,32.812,156.025
C04306=1066.828,322.249,401.075,174.207,32.807,156.024
C04307=1066.822,322.002,401.108,174.204,32.803,156.023
C04308=1066.816,321.754,401.142,174.201,32.798,156.022
C04309=1066.809,321.506,401.175,174.197,32.793,156.021
C04310=1066.803,321.259,401.209,174.194,32.789,156.020
C04311=1066.797,321.011,401.242,174.191,32.784,156.019
C04312=1066.791,320.763,401.276,174.188,32.779,156.018
C04313=1066.784,320.516,401.309,174.184,32.775,156.017
C04314=1066.779,320.268,401.343,174.181,32.770,156.017
C04315=1066.772,320.020,401.376,174.178,32.766,156.016
C04316=1066.766,319.772,401.409,174.174,32.761,156.015
C04317=1066.759,319.525,401.443,174.171,32.757,156.014
C04318=1066.754,319.277,401.476,174.168,32.752,156.013
C04319=1066.747,319.029,401.509,174.165,32.748,156.012
C04320=1066.741,318.782,401.543,174.161,32.743,156.011
C04321=1066.736,318.548,401.574,174.158,32.739,156.010
C04322=1066.730,318.315,401.606,174.155,32.734,156.010
C04323=1066.724,318.081,401.637,174.152,32.730,156.009
C04324=1066.718,317.848,401.669,174.149,32.725,156.008
C04325=1066.712,317.615,401.699,174.146,32.721,156.007
C04326=1066.707,317.381,401.731,174.143,32.717,156.006
C04327=1066.701,317.148,401.762,174.140,32.713,156.005
C04328=1066.695,316.915,401.794,174.137,32.709,156.005
C04329=1066.688,316.667,401.827,174.134,32.704,156.004
C04330=1066.682,316.419,401.860,174.130,32.699,156.003
C04331=1066.676,316.171,401.893,174.127,32.695,156.002
C04332=1066.671,315.923,401.926,174.124,32.690,156.001
C04333=1066.664,315.676,401.959,174.121,32.686,156.000
C04334=1066.659,315.428,401.992,174.118,32.681,155.999
C04335=1066.652,315.180,402.025,174.114,32.677,155.998
C04336=1066.646,314.933,402.058,174.112,32.672,155.998
C04337=1066.640,314.685,402.092,174.109,32.667,155.997
C04338=1066.634,314.438,402.125,174.106,32.663,155.996
C04339=1066.628,314.190,402.157,174.103,32.658,155.995
C04340=1066.622,313.942,402.191,174.099,32.654,155.994
C04341=1066.615,313.694,402.224,174.096,32.650,155.993
C04342=1066.609,313.446,402.255,174.093,32.645,155.992
C04343=1066.602,313.198,402.288,174.090,32.641,155.992
C04344=1066.596,312.951,402.321,174.086,32.636,155.991
C04345=1066.590,312.703,402.353,174.083,32.632,155.990
C04346=1066.583,312.456,402.386,174.080,32.628,155.989
C04347=1066.577,312.207,402.419,174.077,32.623,155.988
C04348=1066.570,311.960,402.452,174.074,32.619,155.987
C04349=1066.564,311.712,402.484,174.070,32.614,155.987
C04350=1066.558,311.464,402.517,174.067,32.610,155.986
C04351=1066.552,311.216,402.550,174.064,32.606,155.985
C04352=1066.545,310.969,402.582,174.061,32.601,155.984
C04353=1066.539,310.721,402.614,174.058,32.597,155.983
C04354=1066.532,310.473,402.646,174.054,32.593,155.982
C04355=1066.526,310.226,402.679,174.051,32.588,155.982
C04356=1066.520,309.978,402.712,174.049,32.584,155.981
C04357=1066.514,309.730,402.744,174.046,32.580,155.980
C04358=1066.507,309.482,402.777,174.043,32.575,155.979
C04359=1066.501,309.235,402.809,174.039,32.571,155.978
C04360=1066.495,308.987,402.841,174.036,32.567,155.977
C04361=1066.488,308.739,402.874,174.033,32.562,155.977
C04362=1066.482,308.491,402.906,174.030,32.558,155.976
C04363=1066.476,308.243,402.938,174.027,32.554,155.975
C04364=1066.470,307.996,402.971,174.024,32.549,155.974
C04365=1066.464,307.748,403.003,174.020,32.545,155.973
C04366=1066.457,307.500,403.036,174.017,32.540,155.972
C04367=1066.451,307.252,403.068,174.014,32.536,155.972
C04368=1066.444,307.005,403.100,174.011,32.532,155.971
C04369=1066.438,306.756,403.132,174.008,32.528,155.970
C04370=1066.432,306.509,403.165,174.005,32.524,155.969
C04371=1066.426,306.260,403.197,174.002,32.519,155.968
C04372=1066.420,306.014,403.229,173.999,32.514,155.967
C04373=1066.414,305.766,403.261,173.996,32.510,155.967
C04374=1066.407,305.518,403.293,173.993,32.506,155.966
C04375=1066.401,305.270,403.325,173.990,32.502,155.965
C04376=1066.395,305.022,403.357,173.987,32.497,155.964
C04377=1066.390,304.790,403.388,173.984,32.493,155.963
C04378=1066.383,304.558,403.418,173.981,32.489,155.963
C04379=1066.378,304.327,403.448,173.978,32.485,155.962
C04380=1066.372,304.096,403.478,173.975,32.481,155.961
C04381=1066.366,303.864,403.507,173.972,32.477,155.960
C04382=1066.360,303.632,403.538,173.969,32.473,155.960
C04383=1066.355,303.401,403.568,173.967,32.469,155.959
C04384=1066.349,303.169,403.597,173.964,32.465,155.958
C04385=1066.343,302.922,403.629,173.961,32.461,155.957
C04386=1066.337,302.673,403.662,173.958,32.457,155.957
C04387=1066.331,302.426,403.693,173.955,32.452,155.956
C04388=1066.325,302.178,403.725,173.952,32.448,155.955
C04389=1066.318,301.930,403.757,173.949,32.444,155.954
C04390=1066.312,301.682,403.789,173.946,32.439,155.953
C04391=1066.307,301.435,403.821,173.943,32.435,155.952
C04392=1066.300,301.187,403.852,173.940,32.431,155.952
C04393=1066.294,300.939,403.884,173.937,32.426,155.951
C04394=1066.288,300.690,403.917,173.934,32.422,155.950
C04395=1066.283,300.443,403.948,173.931,32.418,155.949
C04396=1066.276,300.196,403.980,173.928,32.414,155.948
C04397=1066.270,299.947,404.012,173.925,32.409,155.948
C04398=1066.264,299.700,404.044,173.922,32.405,155.947
C04399=1066.258,299.452,404.075,173.920,32.401,155.946
C04400=1066.252,299.204,404.107,173.917,32.397,155.945
C04401=1066.246,298.956,404.139,173.914,32.392,155.944
C04402=1066.240,298.708,404.171,173.911,32.388,155.944
C04403=1066.234,298.460,404.203,173.908,32.384,155.943
C04404=1066.228,298.213,404.234,173.905,32.379,155.942
C04405=1066.222,297.964,404.266,173.902,32.375,155.941
C04406=1066.216,297.717,404.297,173.898,32.371,155.940
C04407=1066.210,297.469,404.329,173.895,32.367,155.940
C04408=1066.204,297.221,404.361,173.892,32.362,155.939
C04409=1066.198,296.973,404.392,173.889,32.358,155.938
C04410=1066.192,296.725,404.424,173.886,32.354,155.937
C04411=1066.186,296.477,404.455,173.884,32.350,155.936
C04412=1066.180,296.230,404.486,173.881,32.345,155.936
C04413=1066.174,295.981,404.518,173.878,32.341,155.935
C04414=1066.167,295.733,404.550,173.875,32.337,155.934
C04415=1066.162,295.485,404.581,173.872,32.333,155.933
C04416=1066.155,295.237,404.612,173.869,32.329,155.932
C04417=1066.149,294.990,404.643,173.866,32.324,155.932
C04418=1066.143,294.742,404.675,173.863,32.320,155.931
C04419=1066.137,294.493,404.706,173.860,32.316,155.930
C04420=1066.130,294.246,404.737,173.857,32.312,155.929
C04421=1066.124,293.998,404.769,173.854,32.308,155.929
C04422=1066.118,293.750,404.800,173.852,32.304,155.928
C04423=1066.112,293.502,404.831,173.849,32.299,155.927
C04424=1066.106,293.254,404.863,173.846,32.295,155.926
C04425=1066.100,293.006,404.893,173.843,32.291,155.925
C04426=1066.093,292.758,404.925,173.840,32.287,155.925
C04427=1066.087,292.510,404.955,173.837,32.283,155.924
C04428=1066.082,292.262,404.987,173.834,32.279,155.923
C04429=1066.075,292.014,405.018,173.831,32.274,155.922
C04430=1066.069,291.767,405.049,173.828,32.271,155.922
C04431=1066.063,291.518,405.081,173.825,32.266,155.921
C04432=1066.057,291.271,405.111,173.824,32.262,155.920
C04433=1066.051,291.047,405.139,173.821,32.258,155.919
C04434=1066.046,290.823,405.167,173.818,32.255,155.919
C04435=1066.040,290.598,405.195,173.815,32.251,155.918
C04436=1066.034,290.374,405.224,173.813,32.247,155.917
C04437=1066.029,290.150,405.251,173.810,32.244,155.917
C04438=1066.024,289.926,405.280,173.807,32.239,155.916
C04439=1066.018,289.702,405.307,173.805,32.236,155.915
C04440=1066.012,289.478,405.335,173.802,32.232,155.914
C04441=1066.007,289.230,405.366,173.799,32.228,155.914
C04442=1066.000,288.982,405.397,173.797,32.224,155.913
C04443=1065.995,288.734,405.428,173.794,32.220,155.912
C04444=1065.988,288.485,405.458,173.791,32.215,155.911
C04445=1065.982,288.238,405.490,173.788,32.212,155.911
C04446=1065.976,287.990,405.520,173.785,32.207,155.910
C04447=1065.970,287.742,405.551,173.783,32.203,155.909
C04448=1065.963,287.493,405.581,173.780,32.200,155.908
C04449=1065.957,287.246,405.612,173.777,32.195,155.908
C04450=1065.951,286.998,405.643,173.774,32.192,155.907
C04451=1065.945,286.750,405.673,173.772,32.187,155.906
C04452=1065.939,286.501,405.704,173.769,32.183,155.905
C04453=1065.933,286.254,405.735,173.766,32.179,155.905
C04454=1065.926,286.006,405.766,173.763,32.175,155.904
C04455=1065.920,285.758,405.796,173.760,32.171,155.903
C04456=1065.914,285.510,405.827,173.757,32.167,155.902
C04457=1065.908,285.261,405.857,173.754,32.163,155.902
C04458=1065.902,285.014,405.888,173.751,32.159,155.901
C04459=1065.896,284.765,405.918,173.749,32.155,155.900
C04460=1065.890,284.517,405.949,173.747,32.150,155.899
C04461=1065.884,284.270,405.980,173.744,32.147,155.899
C04462=1065.877,284.022,406.011,173.741,32.142,155.898
C04463=1065.872,283.774,406.041,173.738,32.138,155.897
C04464=1065.866,283.526,406.071,173.735,32.134,155.896
C04465=1065.859,283.277,406.102,173.732,32.130,155.896
C04466=1065.854,283.030,406.132,173.729,32.126,155.895
C04467=1065.846,282.781,406.162,173.726,32.122,155.894
C04468=1065.841,282.534,406.193,173.725,32.118,155.893
C04469=1065.835,282.286,406.223,173.722,32.114,155.893
C04470=1065.828,282.037,406.254,173.719,32.110,155.892
C04471=1065.823,281.789,406.284,173.716,32.105,155.891
C04472=1065.817,281.541,406.314,173.713,32.102,155.890
C04473=1065.811,281.293,406.344,173.710,32.097,155.890
C04474=1065.805,281.045,406.375,173.707,32.093,155.889
C04475=1065.799,280.797,406.405,173.705,32.089,155.888
C04476=1065.793,280.549,406.436,173.702,32.085,155.887
C04477=1065.787,280.300,406.466,173.700,32.081,155.886
C04478=1065.780,280.053,406.496,173.697,32.077,155.886
C04479=1065.775,279.804,406.526,173.694,32.073,155.885
C04480=1065.769,279.557,406.556,173.691,32.069,155.884
C04481=1065.762,279.308,406.587,173.688,32.065,155.883
C04482=1065.756,279.061,406.617,173.686,32.061,155.883
C04483=1065.750,278.812,406.646,173.683,32.057,155.882
C04484=1065.744,278.564,406.677,173.681,32.053,155.881
C04485=1065.737,278.316,406.707,173.678,32.049,155.881
C04486=1065.732,278.068,406.737,173.675,32.045,155.880
C04487=1065.726,277.820,406.767,173.672,32.041,155.879
C04488=1065.720,277.571,406.797,173.670,32.037,155.878
C04489=1065.714,277.353,406.823,173.667,32.033,155.878
C04490=1065.709,277.134,406.849,173.665,32.030,155.877
C04491=1065.703,276.915,406.877,173.662,32.026,155.876
C04492=1065.698,276.697,406.903,173.660,32.023,155.876
C04493=1065.693,276.477,406.929,173.658,32.019,155.875
C04494=1065.688,276.258,406.956,173.656,32.015,155.874
C04495=1065.682,276.040,406.982,173.653,32.012,155.874
C04496=1065.676,275.821,407.008,173.651,32.009,155.873
C04497=1065.671,275.573,407.038,173.648,32.004,155.872
C04498=1065.665,275.325,407.068,173.645,32.001,155.872
C04499=1065.658,275.076,407.098,173.642,31.996,155.871
C04500=1065.652,274.828,407.128,173.641,31.993,155.870
C04501=1065.646,274.580,407.157,173.638,31.988,155.869
C04502=1065.640,274.332,407.187,173.635,31.984,155.869
C04503=1065.635,274.084,407.217,173.632,31.980,155.868
C04504=1065.628,273.836,407.247,173.629,31.976,155.867
C04505=1065.622,273.587,407.277,173.627,31.972,155.867
C04506=1065.616,273.340,407.307,173.624,31.968,155.866
C04507=1065.610,273.091,407.336,173.621,31.964,155.865
C04508=1065.604,272.843,407.366,173.619,31.960,155.864
C04509=1065.598,272.595,407.396,173.616,31.956,155.864
C04510=1065.592,272.347,407.425,173.614,31.952,155.863
C04511=1065.586,272.099,407.454,173.611,31.948,155.862
C04512=1065.579,271.850,407.484,173.608,31.944,155.861
C04513=1065.574,271.602,407.514,173.605,31.940,155.861
C04514=1065.567,271.354,407.543,173.603,31.936,155.860
C04515=1065.561,271.106,407.573,173.601,31.932,155.859
C04516=1065.555,270.858,407.602,173.598,31.928,155.859
C04517=1065.550,270.609,407.632,173.595,31.924,155.858
C04518=1065.543,270.361,407.661,173.592,31.920,155.857
C04519=1065.537,270.114,407.691,173.590,31.916,155.856
C04520=1065.531,269.865,407.720,173.587,31.912,155.856
C04521=1065.525,269.617,407.750,173.585,31.908,155.855
C04522=1065.520,269.369,407.779,173.582,31.904,155.854
C04523=1065.513,269.120,407.809,173.580,31.901,155.853
C04524=1065.506,268.872,407.838,173.577,31.896,155.853
C04525=1065.501,268.624,407.868,173.574,31.892,155.852
C04526=1065.494,268.376,407.897,173.572,31.888,155.851
C04527=1065.488,268.128,407.926,173.569,31.884,155.850
C04528=1065.483,267.879,407.956,173.567,31.881,155.850
C04529=1065.476,267.631,407.985,173.564,31.876,155.849
C04530=1065.470,267.383,408.014,173.562,31.873,155.848
C04531=1065.464,267.135,408.043,173.559,31.868,155.848
C04532=1065.458,266.887,408.072,173.556,31.865,155.847
C04533=1065.452,266.638,408.101,173.553,31.860,155.846
C04534=1065.446,266.390,408.131,173.551,31.857,155.845
C04535=1065.440,266.142,408.160,173.549,31.853,155.845
C04536=1065.434,265.894,408.189,173.546,31.848,155.844
C04537=1065.428,265.646,408.218,173.544,31.845,155.843
C04538=1065.422,265.397,408.247,173.541,31.840,155.843
C04539=1065.416,265.149,408.277,173.538,31.837,155.842
C04540=1065.410,264.901,408.306,173.535,31.832,155.841
C04541=1065.404,264.653,408.335,173.534,31.829,155.840
C04542=1065.397,264.405,408.364,173.531,31.825,155.840
C04543=1065.392,264.156,408.394,173.528,31.821,155.839
C04544=1065.386,263.908,408.423,173.526,31.817,155.838
C04545=1065.381,263.690,408.448,173.523,31.813,155.838
C04546=1065.375,263.474,408.473,173.521,31.809,155.837
C04547=1065.370,263.257,408.499,173.519,31.806,155.836
C04548=1065.364,263.040,408.523,173.517,31.803,155.836
C04549=1065.359,262.823,408.549,173.515,31.800,155.835
C04550=1065.353,262.606,408.574,173.512,31.796,155.835
C04551=1065.348,262.389,408.600,173.510,31.793,155.834
C04552=1065.342,262.171,408.624,173.508,31.790,155.833
C04553=1065.336,261.923,408.653,173.505,31.785,155.833
C04554=1065.330,261.675,408.682,173.502,31.781,155.832
C04555=1065.324,261.426,408.711,173.501,31.778,155.831
C04556=1065.317,261.178,408.740,173.498,31.773,155.830
C04557=1065.311,260.930,408.769,173.495,31.770,155.830
C04558=1065.305,260.681,408.797,173.493,31.766,155.829
C04559=1065.299,260.433,408.826,173.490,31.762,155.828
C04560=1065.293,260.186,408.855,173.487,31.758,155.828
C04561=1065.287,259.937,408.883,173.486,31.754,155.827
C04562=1065.281,259.689,408.912,173.483,31.750,155.826
C04563=1065.274,259.441,408.940,173.480,31.746,155.825
C04564=1065.268,259.192,408.969,173.478,31.742,155.825
C04565=1065.262,258.944,408.998,173.475,31.739,155.824
C04566=1065.256,258.696,409.026,173.472,31.734,155.823
C04567=1065.250,258.447,409.055,173.471,31.731,155.823
C04568=1065.244,258.199,409.084,173.468,31.727,155.822
C04569=1065.238,257.951,409.113,173.465,31.723,155.821
C04570=1065.232,257.702,409.141,173.463,31.719,155.821
C04571=1065.225,257.455,409.169,173.460,31.715,155.820
C04572=1065.219,257.206,409.197,173.457,31.711,155.819
C04573=1065.213,256.958,409.226,173.456,31.707,155.818
C04574=1065.207,256.709,409.255,173.453,31.703,155.818
C04575=1065.201,256.461,409.284,173.450,31.699,155.817
C04576=1065.195,256.213,409.312,173.448,31.695,155.816
C04577=1065.189,255.965,409.341,173.445,31.691,155.816
C04578=1065.183,255.716,409.369,173.444,31.687,155.815
C04579=1065.177,255.468,409.397,173.441,31.683,155.814
C04580=1065.170,255.219,409.426,173.438,31.679,155.813
C04581=1065.165,254.971,409.454,173.436,31.675,155.813
C04582=1065.159,254.723,409.483,173.433,31.671,155.812
C04583=1065.153,254.474,409.511,173.430,31.668,155.811
C04584=1065.146,254.226,409.539,173.429,31.663,155.811
C04585=1065.140,253.978,409.568,173.426,31.660,155.810
C04586=1065.135,253.730,409.596,173.424,31.656,155.809
C04587=1065.129,253.481,409.624,173.421,31.652,155.808
C04588=1065.123,253.232,409.653,173.418,31.648,155.808
C04589=1065.117,252.985,409.681,173.416,31.644,155.807
C04590=1065.110,252.736,409.709,173.414,31.640,155.806
C04591=1065.104,252.488,409.737,173.412,31.636,155.806
C04592=1065.098,252.239,409.766,173.409,31.632,155.805
C04593=1065.093,251.992,409.794,173.406,31.628,155.804
C04594=1065.087,251.743,409.823,173.404,31.624,155.803
C04595=1065.080,251.494,409.850,173.402,31.620,155.803
C04596=1065.075,251.246,409.878,173.400,31.616,155.802
C04597=1065.069,250.998,409.907,173.397,31.612,155.801
C04598=1065.063,250.749,409.936,173.395,31.608,155.801
C04599=1065.057,250.502,409.963,173.392,31.604,155.800
C04600=1065.051,250.253,409.991,173.389,31.600,155.799
C04601=1065.046,250.035,410.016,173.388,31.596,155.798
C04602=1065.040,249.816,410.041,173.386,31.593,155.798
C04603=1065.035,249.599,410.065,173.384,31.589,155.797
C04604=1065.030,249.380,410.090,173.381,31.586,155.797
C04605=1065.025,249.162,410.115,173.379,31.583,155.796
C04606=1065.020,248.943,410.140,173.377,31.579,155.795
C04607=1065.014,248.726,410.164,173.376,31.575,155.795
C04608=1065.009,248.507,410.189,173.374,31.572,155.794
C04609=1065.004,248.259,410.217,173.371,31.568,155.793
C04610=1064.998,248.010,410.246,173.368,31.564,155.793
C04611=1064.992,247.763,410.273,173.366,31.560,155.792
C04612=1064.986,247.514,410.301,173.364,31.556,155.791
C04613=1064.980,247.265,410.330,173.362,31.552,155.790
C04614=1064.974,247.017,410.357,173.359,31.548,155.790
C04615=1064.968,246.769,410.385,173.357,31.544,155.789
C04616=1064.962,246.521,410.413,173.354,31.540,155.788
C04617=1064.956,246.272,410.440,173.353,31.536,155.788
C04618=1064.951,246.024,410.468,173.350,31.532,155.787
C04619=1064.944,245.775,410.496,173.348,31.528,155.786
C04620=1064.938,245.526,410.524,173.345,31.524,155.785
C04621=1064.932,245.279,410.552,173.343,31.520,155.785
C04622=1064.926,245.030,410.580,173.341,31.516,155.784
C04623=1064.920,244.782,410.607,173.339,31.512,155.783
C04624=1064.914,244.533,410.635,173.336,31.508,155.783
C04625=1064.908,244.285,410.662,173.333,31.504,155.782
C04626=1064.902,244.036,410.691,173.331,31.500,155.781
C04627=1064.895,243.788,410.718,173.329,31.496,155.780
C04628=1064.890,243.540,410.746,173.327,31.492,155.780
C04629=1064.884,243.291,410.773,173.324,31.488,155.779
C04630=1064.878,243.043,410.801,173.322,31.484,155.778
C04631=1064.872,242.794,410.829,173.319,31.480,155.778
C04632=1064.866,242.546,410.857,173.318,31.476,155.777
C04633=1064.860,242.297,410.884,173.315,31.472,155.776
C04634=1064.855,242.049,410.912,173.313,31.468,155.775
C04635=1064.848,241.801,410.940,173.310,31.464,155.775
C04636=1064.842,241.552,410.966,173.308,31.460,155.774
C04637=1064.836,241.304,410.995,173.306,31.456,155.773
C04638=1064.831,241.055,411.021,173.304,31.453,155.773
C04639=1064.824,240.807,411.049,173.301,31.448,155.772
C04640=1064.818,240.559,411.076,173.299,31.445,155.771
C04641=1064.812,240.310,411.104,173.296,31.441,155.771
C04642=1064.806,240.062,411.131,173.295,31.436,155.770
C04643=1064.800,239.813,411.158,173.292,31.433,155.769
C04644=1064.794,239.565,411.186,173.290,31.429,155.768
C04645=1064.788,239.316,411.213,173.287,31.425,155.768
C04646=1064.782,239.068,411.241,173.285,31.421,155.767
C04647=1064.775,238.819,411.268,173.284,31.417,155.766
C04648=1064.769,238.571,411.295,173.281,31.413,155.765
C04649=1064.764,238.322,411.323,173.279,31.409,155.765
C04650=1064.758,238.074,411.350,173.276,31.405,155.764
C04651=1064.751,237.825,411.377,173.274,31.401,155.763
C04652=1064.745,237.577,411.404,173.272,31.397,155.763
C04653=1064.739,237.328,411.431,173.270,31.393,155.762
C04654=1064.734,237.080,411.459,173.267,31.389,155.761
C04655=1064.727,236.831,411.486,173.265,31.385,155.761
C04656=1064.721,236.583,411.513,173.263,31.381,155.760
C04657=1064.715,236.362,411.538,173.261,31.378,155.759
C04658=1064.711,236.141,411.562,173.259,31.374,155.759
C04659=1064.705,235.919,411.586,173.257,31.370,155.758
C04660=1064.700,235.698,411.610,173.255,31.367,155.757
C04661=1064.695,235.476,411.635,173.253,31.363,155.757
C04662=1064.689,235.255,411.659,173.251,31.360,155.756
C04663=1064.684,235.034,411.683,173.249,31.356,155.755
C04664=1064.678,234.812,411.707,173.247,31.353,155.755
C04665=1064.673,234.564,411.734,173.244,31.348,155.754
C04666=1064.667,234.316,411.761,173.243,31.345,155.753
C04667=1064.660,234.067,411.788,173.241,31.341,155.753
C04668=1064.655,233.819,411.815,173.238,31.337,155.752
C04669=1064.649,233.570,411.842,173.236,31.333,155.751
C04670=1064.642,233.322,411.869,173.233,31.329,155.750
C04671=1064.636,233.073,411.896,173.232,31.325,155.750
C04672=1064.630,232.824,411.923,173.230,31.321,155.749
C04673=1064.624,232.576,411.950,173.227,31.317,155.748
C04674=1064.619,232.328,411.976,173.225,31.313,155.748
C04675=1064.613,232.078,412.004,173.223,31.309,155.747
C04676=1064.607,231.831,412.031,173.221,31.305,155.746
C04677=1064.601,231.582,412.058,173.218,31.301,155.745
C04678=1064.595,231.333,412.085,173.216,31.297,155.745
C04679=1064.589,231.085,412.112,173.214,31.293,155.744
C04680=1064.583,230.836,412.138,173.212,31.289,155.743
C04681=1064.577,230.588,412.165,173.210,31.285,155.743
C04682=1064.571,230.339,412.192,173.207,31.281,155.742
C04683=1064.565,230.091,412.218,173.205,31.277,155.741
C04684=1064.559,229.842,412.245,173.204,31.273,155.740
C04685=1064.552,229.594,412.272,173.201,31.269,155.740
C04686=1064.546,229.346,412.299,173.199,31.265,155.739
C04687=1064.541,229.097,412.325,173.196,31.261,155.738
C04688=1064.534,228.848,412.352,173.194,31.257,155.738
C04689=1064.529,228.599,412.379,173.193,31.253,155.737
C04690=1064.523,228.351,412.405,173.190,31.249,155.736
C04691=1064.516,228.103,412.431,173.188,31.245,155.736
C04692=1064.510,227.854,412.458,173.185,31.241,155.735
C04693=1064.504,227.606,412.485,173.184,31.237,155.734
C04694=1064.498,227.357,412.512,173.182,31.233,155.733
C04695=1064.493,227.109,412.538,173.179,31.229,155.733
C04696=1064.486,226.860,412.565,173.177,31.225,155.732
C04697=1064.480,226.612,412.591,173.176,31.221,155.731
C04698=1064.474,226.363,412.618,173.173,31.217,155.731
C04699=1064.468,226.115,412.645,173.171,31.213,155.730
C04700=1064.461,225.866,412.670,173.168,31.209,155.729
C04701=1064.456,225.617,412.697,173.167,31.205,155.728
C04702=1064.450,225.369,412.724,173.165,31.201,155.728
C04703=1064.444,225.121,412.750,173.162,31.197,155.727
C04704=1064.438,224.872,412.777,173.160,31.193,155.726
C04705=1064.431,224.623,412.803,173.158,31.189,155.726
C04706=1064.426,224.374,412.829,173.156,31.185,155.725
C04707=1064.420,224.126,412.856,173.154,31.181,155.724
C04708=1064.414,223.878,412.882,173.152,31.177,155.723
C04709=1064.408,223.630,412.909,173.149,31.173,155.723
C04710=1064.402,223.381,412.934,173.148,31.169,155.722
C04711=1064.396,223.132,412.961,173.146,31.165,155.721
C04712=1064.390,222.883,412.988,173.143,31.161,155.721
C04713=1064.385,222.658,413.011,173.141,31.157,155.720
C04714=1064.379,222.432,413.035,173.140,31.153,155.719
C04715=1064.374,222.207,413.060,173.138,31.150,155.719
C04716=1064.369,221.982,413.083,173.136,31.146,155.718
C04717=1064.363,221.756,413.107,173.134,31.143,155.717
C04718=1064.358,221.531,413.131,173.133,31.139,155.717
C04719=1064.352,221.306,413.154,173.131,31.135,155.716
C04720=1064.346,221.080,413.178,173.128,31.132,155.715
C04721=1064.341,220.832,413.205,173.126,31.128,155.715
C04722=1064.334,220.583,413.230,173.124,31.124,155.714
C04723=1064.329,220.335,413.257,173.122,31.120,155.713
C04724=1064.322,220.087,413.283,173.120,31.115,155.712
C04725=1064.317,219.838,413.309,173.118,31.112,155.712
C04726=1064.310,219.590,413.335,173.116,31.107,155.711
C04727=1064.304,219.340,413.361,173.114,31.103,155.710
C04728=1064.298,219.092,413.387,173.112,31.100,155.710
C04729=1064.292,218.843,413.413,173.110,31.095,155.709
C04730=1064.286,218.595,413.439,173.108,31.092,155.708
C04731=1064.280,218.346,413.465,173.106,31.087,155.707
C04732=1064.274,218.098,413.491,173.104,31.084,155.707
C04733=1064.268,217.849,413.517,173.101,31.079,155.706
C04734=1064.262,217.601,413.543,173.100,31.075,155.705
C04735=1064.256,217.352,413.569,173.098,31.071,155.705
C04736=1064.250,217.103,413.594,173.095,31.067,155.704
C04737=1064.243,216.855,413.620,173.093,31.063,155.703
C04738=1064.238,216.606,413.646,173.092,31.059,155.702
C04739=1064.231,216.358,413.672,173.090,31.056,155.702
C04740=1064.225,216.109,413.699,173.087,31.051,155.701
C04741=1064.219,215.860,413.724,173.085,31.047,155.700
C04742=1064.213,215.612,413.751,173.084,31.043,155.700
C04743=1064.207,215.363,413.776,173.081,31.039,155.699
C04744=1064.202,215.114,413.802,173.079,31.035,155.698
C04745=1064.195,214.866,413.828,173.077,31.031,155.697
C04746=1064.190,214.617,413.854,173.076,31.027,155.697
C04747=1064.184,214.368,413.879,173.073,31.022,155.696
C04748=1064.178,214.121,413.905,173.071,31.019,155.695
C04749=1064.172,213.872,413.931,173.069,31.014,155.694
C04750=1064.166,213.623,413.956,173.068,31.011,155.694
C04751=1064.161,213.374,413.982,173.065,31.006,155.693
C04752=1064.154,213.126,414.008,173.063,31.002,155.692
C04753=1064.148,212.878,414.034,173.062,30.998,155.692
C04754=1064.142,212.629,414.059,173.059,30.994,155.691
C04755=1064.136,212.380,414.085,173.057,30.990,155.690
C04756=1064.130,212.131,414.110,173.055,30.986,155.689
C04757=1064.124,211.883,414.137,173.054,30.982,155.689
C04758=1064.118,211.634,414.162,173.051,30.978,155.688
C04759=1064.112,211.386,414.187,173.049,30.974,155.687
C04760=1064.106,211.137,414.213,173.047,30.969,155.686
C04761=1064.100,210.888,414.239,173.046,30.966,155.686
C04762=1064.094,210.639,414.264,173.043,30.961,155.685
C04763=1064.088,210.391,414.289,173.041,30.958,155.684
C04764=1064.082,210.142,414.316,173.040,30.953,155.684
C04765=1064.076,209.894,414.341,173.038,30.950,155.683
C04766=1064.069,209.645,414.367,173.036,30.945,155.682
C04767=1064.064,209.397,414.392,173.033,30.941,155.681
C04768=1064.058,209.148,414.417,173.032,30.937,155.681
C04769=1064.052,208.925,414.440,173.030,30.933,155.680
C04770=1064.047,208.702,414.463,173.028,30.930,155.679
C04771=1064.041,208.479,414.485,173.026,30.926,155.679
C04772=1064.036,208.256,414.508,173.025,30.922,155.678
C04773=1064.031,208.033,414.531,173.023,30.919,155.677
C04774=1064.025,207.810,414.554,173.021,30.915,155.677
C04775=1064.020,207.587,414.576,173.019,30.911,155.676
C04776=1064.014,207.364,414.599,173.018,30.908,155.675
C04777=1063.990,206.317,414.703,172.853,30.827,155.669
C04778=1063.984,206.068,414.728,172.852,30.824,155.668
C04779=1063.978,205.820,414.751,172.849,30.821,155.668
C04780=1063.972,205.571,414.777,172.847,30.818,155.667
C04781=1063.967,205.323,414.801,172.844,30.815,155.667
C04782=1063.961,205.073,414.825,172.843,30.812,155.666
C04783=1063.956,204.825,414.850,172.840,30.808,155.666
C04784=1063.950,204.575,414.874,172.838,30.805,155.665
C04785=1063.943,204.328,414.899,172.835,30.802,155.665
C04786=1063.937,204.079,414.923,172.834,30.799,155.664
C04787=1063.932,203.830,414.948,172.832,30.795,155.664
C04788=1063.926,203.581,414.972,172.829,30.792,155.663
C04789=1063.921,203.332,414.996,172.827,30.789,155.663
C04790=1063.914,203.084,415.021,172.825,30.786,155.662
C04791=1063.909,202.835,415.045,172.823,30.783,155.662
C04792=1063.903,202.587,415.070,172.820,30.780,155.661
C04793=1063.898,202.337,415.094,172.818,30.776,155.661
C04794=1063.892,202.089,415.119,172.816,30.773,155.660
C04795=1063.886,201.840,415.143,172.814,30.770,155.660
C04796=1063.880,201.591,415.167,172.811,30.767,155.659
C04797=1063.874,201.342,415.191,172.809,30.764,155.659
C04798=1063.868,201.094,415.215,172.807,30.760,155.658
C04799=1063.862,200.845,415.239,172.805,30.758,155.658
C04800=1063.856,200.596,415.263,172.803,30.755,155.657
C04801=1063.850,200.347,415.287,172.800,30.751,155.657
C04802=1063.844,200.098,415.312,172.798,30.749,155.656
C04803=1063.838,199.850,415.335,172.796,30.745,155.656
C04804=1063.833,199.601,415.360,172.794,30.742,155.655
C04805=1063.826,199.353,415.384,172.791,30.739,155.655
C04806=1063.821,199.103,415.408,172.789,30.736,155.654
C04807=1063.815,198.855,415.432,172.788,30.733,155.654
C04808=1063.809,198.606,415.457,172.785,30.730,155.653
C04809=1063.803,198.357,415.480,172.783,30.727,155.653
C04810=1063.797,198.109,415.504,172.780,30.723,155.652
C04811=1063.791,197.859,415.528,172.779,30.721,155.652
C04812=1063.786,197.611,415.552,172.776,30.717,155.651
C04813=1063.780,197.362,415.576,172.774,30.714,155.651
C04814=1063.774,197.113,415.600,172.772,30.712,155.650
C04815=1063.768,196.865,415.624,172.770,30.708,155.650
C04816=1063.762,196.616,415.649,172.768,30.705,155.649
C04817=1063.756,196.367,415.672,172.765,30.702,155.649
C04818=1063.751,196.118,415.696,172.763,30.699,155.648
C04819=1063.744,195.869,415.720,172.762,30.696,155.648
C04820=1063.739,195.620,415.744,172.759,30.693,155.647
C04821=1063.733,195.372,415.768,172.757,30.690,155.647
C04822=1063.727,195.123,415.792,172.754,30.686,155.646
C04823=1063.721,194.874,415.815,172.753,30.684,155.646
C04824=1063.716,194.625,415.840,172.751,30.681,155.645
C04825=1063.710,194.377,415.863,172.748,30.677,155.645
C04826=1063.704,194.128,415.887,172.746,30.675,155.644
C04827=1063.698,193.879,415.911,172.744,30.671,155.644
C04828=1063.692,193.631,415.934,172.742,30.668,155.643
C04829=1063.686,193.381,415.959,172.740,30.665,155.643
C04830=1063.681,193.133,415.982,172.737,30.662,155.642
C04831=1063.675,192.884,416.006,172.736,30.659,155.642
C04832=1063.669,192.636,416.030,172.734,30.656,155.642
C04833=1063.664,192.386,416.054,172.731,30.653,155.641
C04834=1063.658,192.137,416.078,172.729,30.650,155.641
C04835=1063.652,191.889,416.100,172.727,30.647,155.640
C04836=1063.647,191.640,416.125,172.725,30.644,155.640
C04837=1063.640,191.391,416.149,172.723,30.641,155.639
C04838=1063.634,191.108,416.175,172.720,30.637,155.638
C04839=1063.627,190.825,416.202,172.718,30.634,155.638
C04840=1063.621,190.542,416.229,172.716,30.630,155.637
C04841=1063.615,190.258,416.256,172.713,30.626,155.637
C04842=1063.609,190.010,416.280,172.711,30.624,155.636
C04843=1063.603,189.761,416.303,172.709,30.620,155.636
C04844=1063.597,189.512,416.327,172.707,30.618,155.635
C04845=1063.592,189.264,416.350,172.705,30.615,155.635
C04846=1063.586,189.015,416.374,172.702,30.611,155.634
C04847=1063.580,188.765,416.398,172.701,30.609,155.634
C04848=1063.574,188.517,416.421,172.699,30.605,155.633
C04849=1063.569,188.268,416.445,172.696,30.602,155.633
C04850=1063.563,188.020,416.469,172.694,30.599,155.633
C04851=1063.557,187.771,416.492,172.693,30.596,155.632
C04852=1063.552,187.522,416.516,172.690,30.593,155.631
C04853=1063.546,187.273,416.539,172.688,30.590,155.631
C04854=1063.540,187.024,416.563,172.686,30.587,155.630
C04855=1063.535,186.775,416.586,172.684,30.584,155.630
C04856=1063.529,186.526,416.609,172.682,30.581,155.630
C04857=1063.524,186.278,416.634,172.680,30.578,155.629
C04858=1063.518,186.029,416.657,172.677,30.575,155.629
C04859=1063.512,185.780,416.680,172.676,30.572,155.628
C04860=1063.507,185.531,416.704,172.674,30.568,155.628
C04861=1063.501,185.282,416.727,172.672,30.566,155.627
C04862=1063.495,185.034,416.750,172.669,30.562,155.627
C04863=1063.490,184.785,416.774,172.668,30.560,155.626
C04864=1063.484,184.536,416.797,172.666,30.557,155.626
C04865=1063.478,184.286,416.820,172.663,30.554,155.625
C04866=1063.472,184.038,416.844,172.661,30.550,155.625
C04867=1063.466,183.789,416.867,172.660,30.548,155.624
C04868=1063.461,183.540,416.890,172.657,30.545,155.624
C04869=1063.454,183.292,416.912,172.655,30.542,155.623
C04870=1063.447,183.043,416.936,172.653,30.539,155.623
C04871=1063.442,182.794,416.959,172.652,30.537,155.623
C04872=1063.436,182.545,416.982,172.649,30.533,155.622
C04873=1063.430,182.296,417.005,172.647,30.530,155.622
C04874=1063.425,182.047,417.028,172.645,30.528,155.621
C04875=1063.419,181.798,417.051,172.643,30.524,155.621
C04876=1063.412,181.549,417.075,172.641,30.522,155.620
C04877=1063.406,181.300,417.098,172.639,30.519,155.620
C04878=1063.400,181.052,417.120,172.636,30.516,155.619
C04879=1063.394,180.803,417.143,172.635,30.513,155.619
C04880=1063.388,180.554,417.166,172.633,30.510,155.618
C04881=1063.383,180.305,417.189,172.631,30.507,155.618
C04882=1063.377,180.056,417.212,172.628,30.504,155.618
C04883=1063.371,179.807,417.235,172.627,30.501,155.617
C04884=1063.366,179.558,417.258,172.625,30.499,155.617
C04885=1063.359,179.310,417.280,172.623,30.496,155.616
C04886=1063.353,179.060,417.303,172.620,30.492,155.616
C04887=1063.347,178.812,417.327,172.619,30.490,155.615
C04888=1063.341,178.563,417.350,172.617,30.487,155.615
C04889=1063.335,178.314,417.373,172.614,30.484,155.614
C04890=1063.330,178.065,417.396,172.612,30.481,155.614
C04891=1063.323,177.817,417.418,172.611,30.478,155.614
C04892=1063.317,177.568,417.441,172.609,30.475,155.613
C04893=1063.312,177.318,417.463,172.606,30.472,155.613
C04894=1063.306,177.069,417.486,172.604,30.470,155.612
C04895=1063.300,176.820,417.509,172.603,30.467,155.612
C04896=1063.295,176.571,417.532,172.601,30.464,155.611
C04897=1063.288,176.323,417.555,172.598,30.461,155.611
C04898=1063.283,176.074,417.578,172.596,30.458,155.610
C04899=1063.277,175.825,417.601,172.595,30.455,155.610
C04900=1063.271,175.576,417.624,172.593,30.453,155.609
C04901=1063.265,175.327,417.646,172.591,30.449,155.609
C04902=1063.259,175.044,417.672,172.588,30.446,155.608
C04903=1063.252,174.760,417.698,172.586,30.442,155.608
C04904=1063.245,174.477,417.724,172.584,30.439,155.607
C04905=1063.238,174.194,417.750,172.581,30.436,155.607
C04906=1063.233,173.944,417.772,172.580,30.433,155.606
C04907=1063.227,173.695,417.795,172.578,30.431,155.606
C04908=1063.221,173.446,417.818,172.576,30.427,155.605
C04909=1063.215,173.198,417.841,172.573,30.424,155.605
C04910=1063.209,172.949,417.863,172.572,30.422,155.605
C04911=1063.204,172.700,417.885,172.570,30.419,155.604
C04912=1063.198,172.451,417.908,172.568,30.416,155.604
C04913=1063.193,172.202,417.931,172.566,30.413,155.603
C04914=1063.186,171.954,417.953,172.564,30.410,155.603
C04915=1063.180,171.705,417.976,172.562,30.407,155.602
C04916=1063.175,171.455,417.998,172.560,30.405,155.602
C04917=1063.169,171.207,418.021,172.558,30.401,155.601
C04918=1063.163,170.958,418.044,172.557,30.399,155.601
C04919=1063.157,170.708,418.066,172.554,30.396,155.601
C04920=1063.152,170.459,418.089,172.552,30.393,155.600
C04921=1063.146,170.211,418.111,172.550,30.390,155.600
C04922=1063.140,169.963,418.134,172.549,30.387,155.599
C04923=1063.135,169.713,418.156,172.547,30.384,155.599
C04924=1063.129,169.464,418.179,172.545,30.381,155.598
C04925=1063.123,169.215,418.201,172.543,30.378,155.598
C04926=1063.117,168.966,418.223,172.541,30.375,155.597
C04927=1063.111,168.717,418.246,172.539,30.373,155.597
C04928=1063.106,168.468,418.268,172.537,30.369,155.596
C04929=1063.101,168.220,418.291,172.536,30.367,155.596
C04930=1063.094,167.971,418.314,172.533,30.364,155.596
C04931=1063.089,167.721,418.336,172.531,30.361,155.595
C04932=1063.083,167.473,418.359,172.529,30.358,155.595
C04933=1063.077,167.224,418.380,172.528,30.355,155.594
C04934=1063.072,166.975,418.403,172.526,30.352,155.594
C04935=1063.066,166.726,418.425,172.524,30.349,155.593
C04936=1063.061,166.477,418.448,172.522,30.346,155.593
C04937=1063.054,166.228,418.471,172.520,30.343,155.592
C04938=1063.049,165.979,418.492,172.518,30.341,155.592
C04939=1063.044,165.730,418.515,172.516,30.337,155.591
C04940=1063.037,165.481,418.537,172.514,30.335,155.591
C04941=1063.032,165.232,418.560,172.513,30.332,155.591
C04942=1063.027,164.984,418.582,172.511,30.329,155.590
C04943=1063.020,164.735,418.604,172.508,30.326,155.590
C04944=1063.015,164.485,418.626,172.506,30.323,155.589
C04945=1063.010,164.236,418.649,172.505,30.320,155.589
C04946=1063.004,163.988,418.671,172.503,30.318,155.588
C04947=1062.998,163.739,418.693,172.501,30.314,155.588
C04948=1062.992,163.490,418.716,172.499,30.312,155.587
C04949=1062.987,163.241,418.737,172.498,30.309,155.587
C04950=1062.981,162.992,418.760,172.496,30.306,155.586
C04951=1062.976,162.743,418.782,172.493,30.303,155.586
C04952=1062.970,162.494,418.803,172.492,30.300,155.586
C04953=1062.964,162.245,418.826,172.490,30.297,155.585
C04954=1062.959,161.996,418.849,172.488,30.294,155.585
C04955=1062.953,161.748,418.871,172.486,30.291,155.584
C04956=1062.948,161.498,418.893,172.485,30.288,155.584
C04957=1062.942,161.249,418.915,172.483,30.286,155.583
C04958=1062.936,161.000,418.937,172.481,30.282,155.583
C04959=1062.931,160.752,418.959,172.478,30.280,155.582
C04960=1062.925,160.502,418.981,172.477,30.277,155.582
C04961=1062.919,160.253,419.003,172.475,30.274,155.582
C04962=1062.912,160.005,419.025,172.473,30.271,155.581
C04963=1062.907,159.756,419.047,172.471,30.268,155.581
C04964=1062.901,159.506,419.068,172.470,30.266,155.580
C04965=1062.895,159.257,419.090,172.468,30.263,155.580
C04966=1062.889,158.974,419.115,172.465,30.260,155.579
C04967=1062.883,158.690,419.141,172.464,30.256,155.579
C04968=1062.876,158.406,419.165,172.461,30.253,155.578
C04969=1062.870,158.122,419.190,172.459,30.250,155.578
C04970=1062.863,157.873,419.212,172.457,30.248,155.577
C04971=1062.857,157.624,419.234,172.456,30.244,155.577
C04972=1062.851,157.376,419.255,172.454,30.242,155.576
C04973=1062.846,157.126,419.277,172.452,30.239,155.576
C04974=1062.840,156.877,419.299,172.450,30.236,155.576
C04975=1062.834,156.628,419.320,172.448,30.233,155.575
C04976=1062.829,156.379,419.343,172.446,30.230,155.575
C04977=1062.822,156.130,419.365,172.444,30.228,155.574
C04978=1062.817,155.882,419.386,172.443,30.225,155.574
C04979=1062.811,155.633,419.408,172.441,30.222,155.573
C04980=1062.805,155.383,419.430,172.439,30.219,155.573
C04981=1062.800,155.135,419.451,172.437,30.216,155.573
C04982=1062.793,154.885,419.473,172.436,30.214,155.572
C04983=1062.787,154.636,419.495,172.434,30.211,155.572
C04984=1062.782,154.388,419.516,172.432,30.208,155.571
C04985=1062.776,154.138,419.538,172.430,30.206,155.571
C04986=1062.770,153.889,419.560,172.428,30.203,155.571
C04987=1062.765,153.641,419.581,172.426,30.199,155.570
C04988=1062.758,153.391,419.603,172.424,30.197,155.570
C04989=1062.752,153.142,419.624,172.422,30.194,155.569
C04990=1062.747,152.894,419.646,172.421,30.191,155.569
C04991=1062.741,152.644,419.668,172.419,30.189,155.568
C04992=1062.736,152.396,419.689,172.417,30.186,155.568
C04993=1062.730,152.146,419.711,172.416,30.183,155.567
C04994=1062.723,151.897,419.732,172.414,30.180,155.567
C04995=1062.718,151.649,419.754,172.412,30.177,155.567
C04996=1062.712,151.399,419.775,172.410,30.175,155.566
C04997=1062.706,151.151,419.797,172.409,30.172,155.566
C04998=1062.700,150.902,419.818,172.407,30.169,155.565
C04999=1062.694,150.652,419.840,172.405,30.166,155.565
C05000=1062.689,150.403,419.861,172.402,30.163,155.564
C05001=1062.683,150.154,419.883,172.401,30.161,155.564
C05002=1062.677,149.905,419.904,172.399,30.158,155.564
C05003=1062.671,149.656,419.925,172.397,30.155,155.563
C05004=1062.666,149.408,419.947,172.395,30.153,155.563
C05005=1062.660,149.158,419.968,172.394,30.150,155.562
C05006=1062.654,148.909,419.989,172.392,30.147,155.562
C05007=1062.648,148.660,420.011,172.390,30.144,155.561
C05008=1062.642,148.411,420.032,172.389,30.141,155.561
C05009=1062.636,148.162,420.053,172.387,30.139,155.561
C05010=1062.630,147.913,420.075,172.385,30.136,155.560
C05011=1062.625,147.664,420.096,172.383,30.133,155.560
C05012=1062.619,147.415,420.117,172.382,30.131,155.559
C05013=1062.613,147.166,420.139,172.380,30.128,155.559
C05014=1062.607,146.917,420.160,172.378,30.125,155.559
C05015=1062.601,146.667,420.181,172.376,30.122,155.558
C05016=1062.596,146.419,420.202,172.375,30.119,155.558
C05017=1062.590,146.170,420.224,172.373,30.117,155.557
C05018=1062.584,145.921,420.245,172.371,30.114,155.557
C05019=1062.577,145.672,420.266,172.369,30.111,155.556
C05020=1062.572,145.423,420.287,172.368,30.109,155.556
C05021=1062.566,145.174,420.309,172.366,30.106,155.556
C05022=1062.560,144.925,420.329,172.363,30.103,155.555
C05023=1062.554,144.676,420.351,172.362,30.100,155.555
C05024=1062.549,144.427,420.372,172.360,30.098,155.554
C05025=1062.543,144.177,420.393,172.358,30.095,155.554
C05026=1062.537,143.929,420.414,172.356,30.092,155.553
C05027=1062.530,143.680,420.435,172.355,30.089,155.553
C05028=1062.525,143.431,420.456,172.353,30.086,155.553
C05029=1062.519,143.182,420.477,172.351,30.084,155.552
C05030=1062.512,142.897,420.501,172.349,30.080,155.552
C05031=1062.506,142.613,420.525,172.348,30.078,155.551
C05032=1062.500,142.329,420.550,172.345,30.074,155.551
C05033=1062.493,142.045,420.574,172.343,30.071,155.550
C05034=1062.487,141.796,420.594,172.342,30.068,155.550
C05035=1062.481,141.547,420.616,172.340,30.066,155.549
C05036=1062.475,141.298,420.636,172.338,30.063,155.549
C05037=1062.470,141.049,420.657,172.336,30.060,155.549
C05038=1062.464,140.800,420.678,172.335,30.057,155.548
C05039=1062.458,140.551,420.700,172.333,30.055,155.548
C05040=1062.453,140.301,420.721,172.331,30.052,155.547
C05041=1062.446,140.053,420.741,172.330,30.049,155.547
C05042=1062.440,139.803,420.762,172.328,30.046,155.546
C05043=1062.435,139.555,420.783,172.326,30.043,155.546
C05044=1062.428,139.305,420.804,172.324,30.041,155.546
C05045=1062.423,139.057,420.825,172.323,30.038,155.545
C05046=1062.417,138.808,420.846,172.321,30.035,155.545
C05047=1062.412,138.558,420.866,172.319,30.033,155.544
C05048=1062.405,138.310,420.887,172.317,30.030,155.544
C05049=1062.399,138.060,420.908,172.316,30.027,155.543
C05050=1062.394,137.811,420.929,172.314,30.025,155.543
C05051=1062.388,137.562,420.949,172.312,30.022,155.543
C05052=1062.382,137.313,420.970,172.311,30.019,155.542
C05053=1062.376,137.064,420.991,172.309,30.017,155.542
C05054=1062.370,136.815,421.012,172.307,30.014,155.541
C05055=1062.365,136.565,421.032,172.305,30.011,155.541
C05056=1062.358,136.317,421.053,172.304,30.008,155.541
C05057=1062.352,136.067,421.074,172.302,30.006,155.540
C05058=1062.347,135.818,421.095,172.300,30.003,155.540
C05059=1062.340,135.569,421.116,172.298,30.000,155.539
C05060=1062.335,135.320,421.136,172.297,29.998,155.539
C05061=1062.330,135.071,421.157,172.295,29.994,155.538
C05062=1062.323,134.822,421.178,172.293,29.992,155.538
C05063=1062.318,134.573,421.198,172.292,29.989,155.538
C05064=1062.312,134.324,421.218,172.290,29.986,155.537
C05065=1062.306,134.074,421.239,172.288,29.984,155.537
C05066=1062.300,133.826,421.260,172.286,29.981,155.536
C05067=1062.294,133.577,421.280,172.285,29.978,155.536
C05068=1062.288,133.327,421.301,172.284,29.976,155.536
C05069=1062.282,133.079,421.321,172.282,29.973,155.535
C05070=1062.277,132.830,421.343,172.280,29.970,155.535
C05071=1062.271,132.580,421.363,172.279,29.968,155.534
C05072=1062.265,132.331,421.383,172.277,29.965,155.534
C05073=1062.260,132.082,421.404,172.275,29.962,155.534
C05074=1062.253,131.833,421.424,172.274,29.960,155.533
C05075=1062.248,131.584,421.446,172.272,29.957,155.533
C05076=1062.242,131.335,421.466,172.270,29.954,155.532
C05077=1062.235,131.086,421.486,172.268,29.951,155.532
C05078=1062.230,130.837,421.506,172.267,29.949,155.531
C05079=1062.224,130.588,421.526,172.265,29.946,155.531
C05080=1062.217,130.338,421.547,172.263,29.943,155.531
C05081=1062.212,130.089,421.567,172.262,29.941,155.530
C05082=1062.206,129.841,421.587,172.260,29.938,155.530
C05083=1062.199,129.592,421.608,172.258,29.935,155.529
C05084=1062.194,129.343,421.629,172.256,29.933,155.529
C05085=1062.188,129.094,421.649,172.255,29.930,155.529
C05086=1062.181,128.844,421.669,172.253,29.927,155.528
C05087=1062.176,128.595,421.690,172.251,29.924,155.528
C05088=1062.170,128.346,421.710,172.249,29.922,155.527
C05089=1062.163,128.097,421.730,172.248,29.920,155.527
C05090=1062.158,127.848,421.750,172.246,29.917,155.527
C05091=1062.152,127.599,421.770,172.244,29.914,155.526
C05092=1062.145,127.349,421.791,172.243,29.912,155.526
C05093=1062.140,127.100,421.811,172.242,29.909,155.525
C05094=1062.133,126.816,421.834,172.239,29.906,155.525
C05095=1062.126,126.531,421.857,172.237,29.903,155.525
C05096=1062.120,126.247,421.880,172.236,29.900,155.524
C05097=1062.113,125.964,421.903,172.234,29.897,155.524
C05098=1062.107,125.715,421.924,172.232,29.894,155.523
C05099=1062.101,125.465,421.944,172.231,29.891,155.523
C05100=1062.095,125.216,421.964,172.229,29.889,155.522
C05101=1062.090,124.967,421.984,172.227,29.886,155.522
C05102=1062.084,124.718,422.004,172.225,29.883,155.522
C05103=1062.077,124.468,422.024,172.224,29.881,155.521
C05104=1062.071,124.219,422.044,172.222,29.878,155.521
C05105=1062.066,123.970,422.064,172.220,29.875,155.520
C05106=1062.060,123.721,422.084,172.219,29.873,155.520
C05107=1062.053,123.472,422.105,172.217,29.870,155.520
C05108=1062.047,123.223,422.125,172.216,29.867,155.519
C05109=1062.042,122.973,422.145,172.214,29.865,155.519
C05110=1062.036,122.725,422.165,172.213,29.862,155.518
C05111=1062.030,122.476,422.184,172.211,29.859,155.518
C05112=1062.024,122.227,422.204,172.209,29.857,155.517
C05113=1062.019,121.977,422.225,172.208,29.854,155.517
C05114=1062.013,121.728,422.245,172.206,29.851,155.517
C05115=1062.007,121.479,422.265,172.204,29.848,155.516
C05116=1062.001,121.230,422.285,172.202,29.846,155.516
C05117=1061.996,120.981,422.305,172.201,29.843,155.515
C05118=1061.990,120.732,422.325,172.199,29.840,155.515
C05119=1061.983,120.483,422.345,172.197,29.838,155.515
C05120=1061.977,120.233,422.365,172.197,29.835,155.514
C05121=1061.972,119.984,422.385,172.195,29.832,155.514
C05122=1061.966,119.735,422.405,172.193,29.830,155.513
C05123=1061.960,119.486,422.425,172.191,29.826,155.513
C05124=1061.954,119.237,422.444,172.190,29.824,155.512
C05125=1061.948,118.988,422.464,172.188,29.821,155.512
C05126=1061.943,118.739,422.485,172.186,29.818,155.512
C05127=1061.937,118.489,422.504,172.185,29.816,155.511
C05128=1061.931,118.240,422.524,172.183,29.813,155.511
C05129=1061.925,117.991,422.544,172.181,29.810,155.510
C05130=1061.920,117.742,422.564,172.180,29.808,155.510
C05131=1061.914,117.493,422.584,172.179,29.805,155.510
C05132=1061.908,117.244,422.604,172.177,29.802,155.509
C05133=1061.902,116.994,422.623,172.175,29.799,155.509
C05134=1061.896,116.746,422.643,172.174,29.797,155.508
C05135=1061.891,116.497,422.664,172.172,29.794,155.508
C05136=1061.885,116.247,422.683,172.170,29.791,155.508
C05137=1061.879,115.998,422.703,172.168,29.789,155.507
C05138=1061.873,115.749,422.723,172.167,29.786,155.507
C05139=1061.868,115.500,422.742,172.166,29.783,155.506
C05140=1061.862,115.251,422.762,172.164,29.781,155.506
C05141=1061.856,115.001,422.782,172.163,29.778,155.505
C05142=1061.850,114.752,422.802,172.161,29.775,155.505
C05143=1061.844,114.503,422.822,172.159,29.772,155.505
C05144=1061.838,114.254,422.842,172.158,29.769,155.504
C05145=1061.832,114.005,422.862,172.156,29.767,155.504
C05146=1061.827,113.755,422.881,172.154,29.764,155.503
C05147=1061.821,113.507,422.901,172.153,29.761,155.503
C05148=1061.815,113.257,422.920,172.152,29.759,155.502
C05149=1061.809,113.008,422.940,172.150,29.756,155.502
C05150=1061.803,112.759,422.959,172.148,29.754,155.502
C05151=1061.797,112.510,422.979,172.146,29.751,155.501
C05152=1061.792,112.261,422.998,172.145,29.748,155.501
C05153=1061.786,112.012,423.018,172.143,29.746,155.501
C05154=1061.780,111.763,423.038,172.141,29.743,155.500
C05155=1061.774,111.513,423.057,172.140,29.740,155.500
C05156=1061.768,111.264,423.077,172.139,29.738,155.499
C05157=1061.763,111.015,423.096,172.137,29.735,155.499
C05158=1061.756,110.730,423.119,172.136,29.732,155.498
C05159=1061.749,110.445,423.141,172.133,29.729,155.498
C05160=1061.741,110.162,423.162,172.131,29.725,155.497
C05161=1061.735,109.877,423.184,172.130,29.723,155.497
C05162=1061.729,109.628,423.204,172.128,29.720,155.497
C05163=1061.723,109.379,423.224,172.126,29.717,155.496
C05164=1061.717,109.129,423.243,172.125,29.715,155.496
C05165=1061.711,108.881,423.263,172.124,29.712,155.495
C05166=1061.705,108.632,423.281,172.122,29.709,155.495
C05167=1061.699,108.382,423.301,172.120,29.707,155.495
C05168=1061.693,108.133,423.321,172.119,29.704,155.494
C05169=1061.687,107.884,423.340,172.117,29.702,155.494
C05170=1061.682,107.634,423.359,172.115,29.699,155.494
C05171=1061.675,107.386,423.379,172.113,29.696,155.493
C05172=1061.669,107.136,423.398,172.113,29.694,155.493
C05173=1061.664,106.887,423.417,172.111,29.691,155.492
C05174=1061.658,106.638,423.437,172.109,29.688,155.492
C05175=1061.652,106.389,423.456,172.108,29.686,155.491
C05176=1061.646,106.140,423.475,172.106,29.683,155.491
C05177=1061.640,105.890,423.494,172.104,29.680,155.491
C05178=1061.634,105.641,423.514,172.103,29.677,155.490
C05179=1061.628,105.392,423.533,172.102,29.675,155.490
C05180=1061.622,105.143,423.552,172.100,29.672,155.489
C05181=1061.616,104.893,423.571,172.098,29.669,155.489
C05182=1061.610,104.644,423.590,172.097,29.667,155.489
C05183=1061.604,104.395,423.610,172.095,29.664,155.488
C05184=1061.599,104.147,423.629,172.093,29.661,155.488
C05185=1061.593,103.897,423.648,172.092,29.659,155.488
C05186=1061.587,103.648,423.667,172.091,29.657,155.487
C05187=1061.581,103.398,423.686,172.089,29.654,155.487
C05188=1061.575,103.150,423.706,172.087,29.651,155.486
C05189=1061.569,102.901,423.725,172.086,29.648,155.486
C05190=1061.563,102.651,423.744,172.084,29.646,155.485
C05191=1061.558,102.402,423.764,172.082,29.643,155.485
C05192=1061.551,102.153,423.782,172.081,29.640,155.485
C05193=1061.546,101.903,423.801,172.080,29.638,155.484
C05194=1061.540,101.654,423.821,172.078,29.635,155.484
C05195=1061.535,101.405,423.840,172.077,29.632,155.483
C05196=1061.528,101.156,423.858,172.075,29.630,155.483
C05197=1061.522,100.907,423.878,172.073,29.627,155.483
C05198=1061.517,100.658,423.897,172.071,29.624,155.482
C05199=1061.510,100.408,423.916,172.071,29.622,155.482
C05200=1061.505,100.159,423.935,172.069,29.619,155.481
C05201=1061.498,99.910,423.954,172.067,29.616,155.481
C05202=1061.492,99.660,423.973,172.066,29.613,155.481
C05203=1061.486,99.411,423.992,172.064,29.611,155.480
C05204=1061.480,99.162,424.011,172.062,29.609,155.480
C05205=1061.474,98.913,424.030,172.061,29.606,155.479
C05206=1061.469,98.664,424.049,172.060,29.603,155.479
C05207=1061.462,98.415,424.067,172.058,29.601,155.479
C05208=1061.457,98.166,424.086,172.056,29.598,155.478
C05209=1061.450,97.916,424.105,172.055,29.595,155.478
C05210=1061.445,97.667,424.124,172.053,29.592,155.477
C05211=1061.438,97.418,424.143,172.051,29.590,155.477
C05212=1061.433,97.168,424.162,172.051,29.588,155.477
C05213=1061.426,96.919,424.180,172.049,29.585,155.476
C05214=1061.421,96.670,424.199,172.047,29.582,155.476
C05215=1061.415,96.421,424.218,172.045,29.580,155.476
C05216=1061.409,96.171,424.237,172.044,29.577,155.475
C05217=1061.403,95.922,424.256,172.042,29.574,155.475
C05218=1061.397,95.673,424.275,172.041,29.572,155.474
C05219=1061.391,95.424,424.293,172.040,29.569,155.474
C05220=1061.386,95.175,424.312,172.038,29.566,155.473
C05221=1061.379,94.926,424.331,172.036,29.563,155.473
C05222=1061.373,94.642,424.353,172.035,29.561,155.473
C05223=1061.365,94.357,424.374,172.033,29.558,155.472
C05224=1061.359,94.072,424.395,172.031,29.555,155.472
C05225=1061.352,93.788,424.416,172.030,29.552,155.471
C05226=1061.347,93.539,424.435,172.028,29.549,155.471
C05227=1061.340,93.289,424.454,172.026,29.546,155.471
C05228=1061.335,93.040,424.473,172.025,29.544,155.470
C05229=1061.329,92.792,424.491,172.023,29.541,155.470
C05230=1061.323,92.542,424.510,172.022,29.538,155.469
C05231=1061.317,92.292,424.529,172.020,29.536,155.469
C05232=1061.311,92.043,424.547,172.019,29.533,155.468
C05233=1061.305,91.795,424.566,172.017,29.530,155.468
C05234=1061.299,91.545,424.585,172.015,29.527,155.468
C05235=1061.294,91.295,424.603,172.015,29.525,155.467
C05236=1061.287,91.046,424.622,172.013,29.522,155.467
C05237=1061.282,90.798,424.641,172.011,29.519,155.466
C05238=1061.276,90.548,424.659,172.010,29.517,155.466
C05239=1061.270,90.299,424.677,172.008,29.515,155.466
C05240=1061.263,90.050,424.696,172.006,29.512,155.465
C05241=1061.257,89.800,424.715,172.005,29.509,155.465
C05242=1061.252,89.551,424.733,172.004,29.507,155.465
C05243=1061.246,89.302,424.751,172.002,29.504,155.464
C05244=1061.239,89.053,424.770,172.000,29.502,155.464
C05245=1061.233,88.803,424.788,171.999,29.499,155.463
C05246=1061.227,88.554,424.807,171.998,29.496,155.463
C05247=1061.222,88.305,424.825,171.996,29.494,155.463
C05248=1061.215,88.056,424.843,171.995,29.491,155.462
C05249=1061.209,87.806,424.862,171.993,29.488,155.462
C05250=1061.203,87.557,424.880,171.991,29.485,155.461
C05251=1061.198,87.308,424.899,171.989,29.483,155.461
C05252=1061.191,87.059,424.918,171.989,29.481,155.461
C05253=1061.185,86.809,424.936,171.987,29.478,155.460
C05254=1061.179,86.561,424.954,171.985,29.475,155.460
C05255=1061.173,86.311,424.972,171.984,29.473,155.459
C05256=1061.168,86.061,424.991,171.982,29.470,155.459
C05257=1061.161,85.812,425.009,171.981,29.468,155.459
C05258=1061.156,85.563,425.027,171.980,29.465,155.458
C05259=1061.149,85.314,425.045,171.978,29.462,155.458
C05260=1061.143,85.064,425.064,171.976,29.460,155.458
C05261=1061.138,84.816,425.083,171.975,29.457,155.457
C05262=1061.132,84.566,425.101,171.973,29.454,155.457
C05263=1061.125,84.317,425.119,171.972,29.452,155.456
C05264=1061.119,84.067,425.137,171.970,29.449,155.456
C05265=1061.113,83.819,425.155,171.969,29.447,155.456
C05266=1061.107,83.569,425.173,171.967,29.444,155.455
C05267=1061.102,83.319,425.192,171.965,29.441,155.455
C05268=1061.096,83.070,425.210,171.965,29.439,155.454
C05269=1061.090,82.821,425.228,171.963,29.436,155.454
C05270=1061.084,82.572,425.247,171.961,29.433,155.454
C05271=1061.078,82.323,425.264,171.960,29.431,155.453
C05272=1061.072,82.073,425.283,171.958,29.428,155.453
C05273=1061.066,81.824,425.301,171.957,29.426,155.452
C05274=1061.060,81.575,425.320,171.956,29.423,155.452
C05275=1061.054,81.325,425.338,171.954,29.420,155.452
C05276=1061.049,81.076,425.355,171.952,29.418,155.451
C05277=1061.042,80.827,425.374,171.950,29.415,155.451
C05278=1061.036,80.577,425.392,171.950,29.412,155.450
C05279=1061.030,80.329,425.410,171.948,29.410,155.450
C05280=1061.024,80.079,425.428,171.946,29.407,155.450
C05281=1061.019,79.830,425.446,171.945,29.404,155.449
C05282=1061.013,79.581,425.465,171.943,29.401,155.449
C05283=1061.007,79.331,425.483,171.942,29.399,155.449
C05284=1061.001,79.082,425.500,171.941,29.397,155.448
C05285=1060.995,78.833,425.519,171.939,29.394,155.448
C05286=1060.988,78.548,425.539,171.937,29.391,155.447
C05287=1060.982,78.264,425.560,171.936,29.388,155.447
C05288=1060.975,77.980,425.581,171.934,29.385,155.446
C05289=1060.968,77.695,425.601,171.932,29.382,155.446
C05290=1060.963,77.446,425.619,171.931,29.379,155.446
C05291=1060.956,77.197,425.637,171.929,29.377,155.445
C05292=1060.950,76.947,425.655,171.927,29.374,155.445
C05293=1060.944,76.698,425.673,171.927,29.372,155.444
C05294=1060.938,76.449,425.690,171.925,29.369,155.444
C05295=1060.932,76.200,425.708,171.923,29.366,155.444
C05296=1060.926,75.951,425.726,171.922,29.363,155.443
C05297=1060.920,75.701,425.744,171.920,29.361,155.443
C05298=1060.914,75.452,425.762,171.919,29.359,155.442
C05299=1060.908,75.202,425.780,171.917,29.356,155.442
C05300=1060.902,74.954,425.798,171.916,29.353,155.442
C05301=1060.896,74.704,425.816,171.914,29.350,155.441
C05302=1060.890,74.455,425.833,171.912,29.348,155.441
C05303=1060.884,74.205,425.851,171.912,29.346,155.441
C05304=1060.877,73.956,425.869,171.910,29.343,155.440
C05305=1060.872,73.707,425.886,171.908,29.340,155.440
C05306=1060.865,73.457,425.905,171.907,29.337,155.439
C05307=1060.860,73.208,425.923,171.905,29.335,155.439
C05308=1060.854,72.959,425.940,171.904,29.333,155.439
C05309=1060.848,72.710,425.958,171.903,29.330,155.438
C05310=1060.842,72.460,425.976,171.901,29.327,155.438
C05311=1060.836,72.211,425.993,171.899,29.324,155.437
C05312=1060.830,71.961,426.011,171.898,29.322,155.437
C05313=1060.824,71.712,426.028,171.897,29.319,155.437
C05314=1060.818,71.463,426.046,171.895,29.317,155.436
C05315=1060.812,71.214,426.065,171.893,29.314,155.436
C05316=1060.806,70.965,426.083,171.892,29.311,155.436
C05317=1060.800,70.716,426.100,171.890,29.309,155.435
C05318=1060.794,70.466,426.117,171.889,29.306,155.435
C05319=1060.788,70.217,426.135,171.888,29.303,155.434
C05320=1060.782,69.967,426.153,171.886,29.301,155.434
C05321=1060.777,69.718,426.171,171.884,29.299,155.434
C05322=1060.770,69.469,426.188,171.883,29.296,155.433
C05323=1060.764,69.220,426.205,171.882,29.293,155.433
C05324=1060.758,68.970,426.223,171.880,29.290,155.432
C05325=1060.753,68.721,426.241,171.879,29.288,155.432
C05326=1060.746,68.472,426.258,171.877,29.286,155.432
C05327=1060.740,68.223,426.276,171.875,29.283,155.431
C05328=1060.734,67.973,426.294,171.875,29.280,155.431
C05329=1060.728,67.724,426.311,171.873,29.278,155.431
C05330=1060.722,67.474,426.329,171.871,29.275,155.430
C05331=1060.717,67.225,426.346,171.870,29.273,155.430
C05332=1060.710,66.975,426.363,171.868,29.270,155.429
C05333=1060.704,66.726,426.380,171.867,29.267,155.429
C05334=1060.698,66.476,426.398,171.865,29.265,155.429
C05335=1060.692,66.228,426.415,171.864,29.262,155.428
C05336=1060.686,65.978,426.433,171.862,29.260,155.428
C05337=1060.680,65.729,426.451,171.861,29.257,155.428
C05338=1060.674,65.480,426.468,171.860,29.254,155.427
C05339=1060.668,65.230,426.486,171.858,29.252,155.427
C05340=1060.662,64.981,426.503,171.856,29.249,155.426
C05341=1060.656,64.731,426.520,171.855,29.247,155.426
C05342=1060.650,64.482,426.538,171.854,29.244,155.426
C05343=1060.644,64.233,426.555,171.852,29.242,155.425
C05344=1060.638,63.984,426.572,171.851,29.239,155.425
C05345=1060.631,63.734,426.590,171.849,29.236,155.425
C05346=1060.626,63.485,426.607,171.847,29.234,155.424
C05347=1060.619,63.235,426.624,171.847,29.232,155.424
C05348=1060.613,62.986,426.642,171.845,29.229,155.423
C05349=1060.607,62.737,426.659,171.843,29.227,155.423
C05350=1060.600,62.453,426.678,171.842,29.223,155.423
C05351=1060.593,62.168,426.698,171.840,29.221,155.422
C05352=1060.586,61.884,426.717,171.838,29.218,155.422
C05353=1060.579,61.600,426.737,171.837,29.215,155.421
C05354=1060.573,61.349,426.754,171.835,29.212,155.421
C05355=1060.567,61.100,426.771,171.833,29.210,155.421
C05356=1060.561,60.851,426.789,171.832,29.207,155.420
C05357=1060.554,60.601,426.806,171.831,29.205,155.420
C05358=1060.548,60.353,426.823,171.829,29.202,155.420
C05359=1060.542,60.103,426.840,171.828,29.200,155.419
C05360=1060.536,59.853,426.857,171.826,29.197,155.419
C05361=1060.529,59.604,426.874,171.824,29.194,155.418
C05362=1060.524,59.355,426.892,171.823,29.192,155.418
C05363=1060.517,59.106,426.909,171.822,29.190,155.418
C05364=1060.512,58.856,426.926,171.820,29.187,155.417
C05365=1060.505,58.607,426.943,171.818,29.185,155.417
C05366=1060.499,58.358,426.959,171.817,29.182,155.417
C05367=1060.493,58.108,426.977,171.816,29.179,155.416
C05368=1060.487,57.859,426.994,171.814,29.177,155.416
C05369=1060.481,57.609,427.011,171.813,29.174,155.416
C05370=1060.475,57.360,427.028,171.811,29.172,155.415
C05371=1060.469,57.111,427.044,171.809,29.169,155.415
C05372=1060.463,56.861,427.062,171.809,29.167,155.414
C05373=1060.457,56.612,427.079,171.807,29.164,155.414
C05374=1060.451,56.363,427.096,171.805,29.161,155.414
C05375=1060.445,56.113,427.113,171.804,29.159,155.413
C05376=1060.439,55.864,427.130,171.802,29.156,155.413
C05377=1060.432,55.615,427.147,171.801,29.154,155.413
C05378=1060.427,55.365,427.164,171.800,29.152,155.412
C05379=1060.420,55.116,427.181,171.798,29.149,155.412
C05380=1060.414,54.868,427.198,171.796,29.146,155.412
C05381=1060.408,54.617,427.215,171.795,29.143,155.411
C05382=1060.402,54.368,427.232,171.794,29.141,155.411
C05383=1060.396,54.119,427.248,171.792,29.139,155.410
C05384=1060.390,53.869,427.266,171.791,29.136,155.410
C05385=1060.384,53.620,427.283,171.789,29.134,155.410
C05386=1060.378,53.371,427.299,171.788,29.131,155.409
C05387=1060.373,53.122,427.316,171.787,29.128,155.409
C05388=1060.366,52.872,427.333,171.785,29.126,155.409
C05389=1060.360,52.623,427.350,171.783,29.124,155.408
C05390=1060.354,52.373,427.367,171.782,29.121,155.408
C05391=1060.348,52.124,427.384,171.781,29.118,155.407
C05392=1060.342,51.874,427.400,171.779,29.115,155.407
C05393=1060.336,51.625,427.418,171.777,29.113,155.407
C05394=1060.330,51.376,427.434,171.776,29.110,155.406
C05395=1060.323,51.127,427.452,171.774,29.108,155.406
C05396=1060.318,50.877,427.468,171.773,29.105,155.406
C05397=1060.312,50.628,427.485,171.772,29.103,155.405
C05398=1060.306,50.379,427.502,171.770,29.100,155.405
C05399=1060.300,50.129,427.518,171.768,29.097,155.404
C05400=1060.294,49.879,427.535,171.767,29.095,155.404
C05401=1060.288,49.630,427.552,171.766,29.093,155.404
C05402=1060.282,49.381,427.568,171.764,29.090,155.403
C05403=1060.276,49.132,427.586,171.763,29.087,155.403
C05404=1060.270,48.882,427.603,171.761,29.085,155.403
C05405=1060.264,48.633,427.619,171.760,29.082,155.402
C05406=1060.258,48.384,427.636,171.759,29.080,155.402
C05407=1060.252,48.134,427.653,171.757,29.077,155.401
C05408=1060.247,47.885,427.669,171.755,29.075,155.401
C05409=1060.241,47.636,427.685,171.754,29.072,155.401
C05410=1060.234,47.386,427.703,171.753,29.069,155.400
C05411=1060.228,47.136,427.719,171.751,29.067,155.400
C05412=1060.223,46.887,427.736,171.750,29.064,155.400
C05413=1060.216,46.638,427.753,171.748,29.062,155.399
C05414=1060.210,46.353,427.772,171.746,29.059,155.399
C05415=1060.203,46.068,427.791,171.745,29.055,155.398
C05416=1060.196,45.784,427.810,171.743,29.053,155.398
C05417=1060.189,45.499,427.829,171.742,29.050,155.398
C05418=1060.183,45.250,427.845,171.740,29.047,155.397
C05419=1060.178,45.000,427.862,171.739,29.045,155.397
C05420=1060.172,44.751,427.878,171.738,29.042,155.396
C05421=1060.166,44.501,427.894,171.736,29.040,155.396
C05422=1060.159,44.252,427.912,171.734,29.037,155.396
C05423=1060.154,44.002,427.929,171.733,29.034,155.395
C05424=1060.148,43.753,427.945,171.732,29.032,155.395
C05425=1060.142,43.504,427.961,171.730,29.029,155.395
C05426=1060.136,43.254,427.977,171.729,29.027,155.394
C05427=1060.130,43.005,427.994,171.727,29.024,155.394
C05428=1060.124,42.756,428.011,171.725,29.022,155.394
C05429=1060.117,42.506,428.027,171.725,29.019,155.393
C05430=1060.112,42.257,428.043,171.723,29.016,155.393
C05431=1060.106,42.007,428.060,171.721,29.014,155.392
C05432=1060.100,41.758,428.076,171.720,29.011,155.392
C05433=1060.094,41.509,428.092,171.718,29.009,155.392
C05434=1060.088,41.259,428.108,171.717,29.007,155.391
C05435=1060.082,41.010,428.125,171.716,29.004,155.391
C05436=1060.075,40.760,428.141,171.714,29.002,155.391
C05437=1060.069,40.511,428.158,171.712,28.999,155.390
C05438=1060.063,40.262,428.175,171.711,28.996,155.390
C05439=1060.057,40.013,428.191,171.710,28.994,155.390
C05440=1060.051,39.763,428.207,171.708,28.991,155.389
C05441=1060.045,39.514,428.223,171.707,28.988,155.389
C05442=1060.039,39.265,428.240,171.705,28.986,155.388
C05443=1060.033,39.015,428.256,171.703,28.984,155.388
C05444=1060.027,38.766,428.272,171.703,28.981,155.388
C05445=1060.021,38.516,428.288,171.701,28.979,155.387
C05446=1060.015,38.267,428.305,171.699,28.976,155.387
C05447=1060.009,38.018,428.321,171.698,28.973,155.387
C05448=1060.003,37.768,428.337,171.696,28.971,155.386
C05449=1059.997,37.518,428.354,171.695,28.968,155.386
C05450=1059.991,37.269,428.370,171.693,28.966,155.386
C05451=1059.985,37.020,428.386,171.692,28.963,155.385
C05452=1059.979,36.770,428.402,171.690,28.961,155.385
C05453=1059.973,36.521,428.417,171.688,28.959,155.385
C05454=1059.967,36.271,428.434,171.688,28.956,155.384
C05455=1059.961,36.022,428.450,171.686,28.954,155.384
C05456=1059.955,35.773,428.466,171.684,28.951,155.383
C05457=1059.949,35.523,428.482,171.683,28.949,155.383
C05458=1059.942,35.274,428.498,171.681,28.946,155.383
C05459=1059.936,35.024,428.515,171.680,28.944,155.382
C05460=1059.930,34.775,428.531,171.679,28.941,155.382
C05461=1059.924,34.526,428.547,171.677,28.939,155.382
